
// ===== library types =====

// folder: Library/Modbus/Core/sb

TYPE "mb_station_block_udt"
   STRUCT
      conf : Struct   // Configuration
         skip_code : Bool;   // Skip all code in header and footer fc.
         disable : Bool;   // Skip all queries
         read_only : Bool;   // Skip all write queries. (fc 5,6,15,16)
         max_comm_error : USInt := 2;   // Repeating erros before communication_error flag is set
         exec_x_quries : USInt := 1;   // Number of queries to be exec. at each loop.
      END_STRUCT;
      out : Struct   // Outputs
         error : Bool;   // All errors, including communication errors
         communication_error : Bool;   // only communication errors
         finnish : Bool;   // qid is handed over to next device.
      END_STRUCT;
      log : Struct   // Logging for development and debugging.
         connected_time : DTL;   // The time the device was connected to the bus
         disconnected_time : DTL;   // The time, if a device was disconnected to the bus
         done_cnt : UDInt;   // Successfully queries counter for this device
         error_comm_cnt : UDInt;   // Communication erros cnt.
         error_exception_cnt : UDInt;   // Failed queries counter for this device
         error_status : Word;   // Status code from mb_master or mb_client
         error_data_addr : UDInt;   // d_addr for last failed querie; handy for troubleshooting
      END_STRUCT;
      z : Struct   // Internal states.
         header_qid : UInt;   // qid value at device header
         comm_err_cnt : USInt;   // Repeating communication errors
         exec_cnt : USInt;   // Numb. of exec. q. this loop
         offset_qid : UInt := 1;   // Device query id.
         err_hold : Bool;   // Help var for .out.error
      END_STRUCT;
   END_STRUCT;
END_TYPE

// folder: Library/Modbus/Station blocks/sb untested/Mettler

TYPE "mettlerToledoInd560Udt"
   STRUCT
      readMsgSlot : Array[1..4] of Struct
         cmdRespons : Struct
            FP_1 : Bool;
            FP_2 : Bool;
            FP_3 : Bool;
            FP_4 : Bool;
            FP_5 : Bool;
            data_integrity : Bool;
            cmdAck1 : Bool;
            cmdAck2 : Bool;
         END_STRUCT;
         reserved : Byte;   // volt
         data : Real;
         scale_status : Struct
            x08_Enter_Key : Bool;
            x09_Input_1 : Bool;
            x10_Input_2 : Bool;
            x11_Input_3 : Bool;
            x12_Motion : Bool;
            x13_Net_Mode : Bool;
            x14_Data_Integrity_2 : Bool;
            x15_Data_OK : Bool;
            x00_Target_1 : Bool;
            x01_Comparator_1 : Bool;
            x02_Targe_2 : Bool;
            x03_Comparator_2 : Bool;
            x04_Target_3 : Bool;
            x05_Alway_true : Bool;
            x06_TE_bit_1 : Bool;
            x07_TE_bit_2 : Bool;
         END_STRUCT;
      END_STRUCT;
      writeMsgSlot : Array[1..4] of Struct
         cmd : UInt;
         data : Real;
      END_STRUCT;
      run : Struct   // Data calculated from readMsgSlot
         PF : Array[1..4] of USInt;   // Floating point input indication
         cmdAck : Array[1..4] of USInt;
      END_STRUCT;
      occupiedMsgSlots : Array[1..4] of Bool;
      queryDone : Struct
         read : Bool;
         write : Bool;
      END_STRUCT;
   END_STRUCT;
END_TYPE

// folder: (top level)

FUNCTION_BLOCK "modbus_rtu_1500"   // FB97, LAD
TITLE = Example modbus rtu for S7-1500
{ S7_Optimized_Access := 'TRUE' }
VERSION : 0.1
   VAR
      mb_master_ctrl : "mb_master_1500_ctrl";
      mb_query : "mb_query";
      aquaMaster_device1 : "abb_aquaMaster_3";
      aquaMaster_device2 : "abb_aquaMaster_3";
      Auma_valve : "Auma_valve";
      Phoenix_Contact_UPS : "Phoenix_Contact_UPS";
   END_VAR
   VAR_TEMP   // added for the SCL form of the ladder/FBD networks
      _w1 : Bool;
   END_VAR
BEGIN

REGION Network 1: Modbus master
   // hardware_id:            Can be found inside "Device configuration". Replace hardware_id with correct id.
   // operating_mode:    0: RS232, 2: RS422, 4: RS485.
   // baud:                         Bits per sec. (Parity is even by default)
   // mb_query:                The FB that connects everything together.
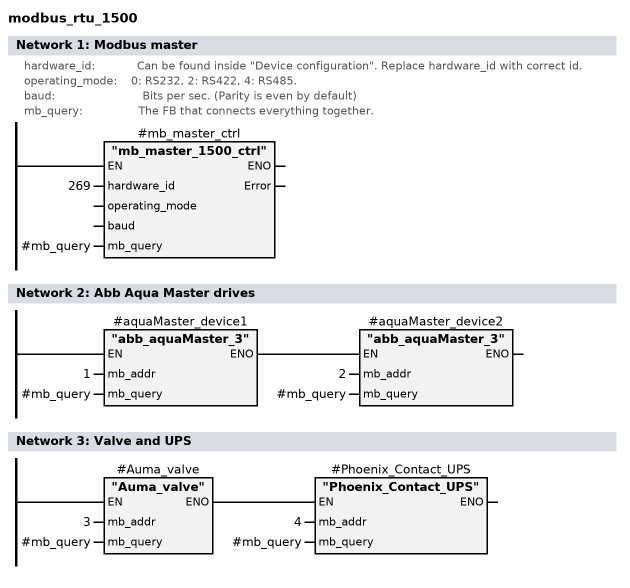
   RUNG wire#powerrail
      #mb_master_ctrl(hardware_id := 269, operating_mode :=, baud :=, mb_query := #mb_query, Error =>)
   END_RUNG
   // the same network as SCL:
   #mb_master_ctrl(hardware_id := 269, mb_query := #mb_query);   // "mb_master_1500_ctrl"
END_REGION

REGION Network 2: Abb Aqua Master drives
   RUNG wire#powerrail
      #aquaMaster_device1(mb_addr := 1, mb_query := #mb_query)
      #aquaMaster_device2(mb_addr := 2, mb_query := #mb_query)
   END_RUNG
   // the same network as SCL:
   #aquaMaster_device1(mb_addr := 1, mb_query := #mb_query, ENO => #_w1);   // "abb_aquaMaster_3"
   IF #_w1 THEN
       #aquaMaster_device2(mb_addr := 2, mb_query := #mb_query);   // "abb_aquaMaster_3"
   END_IF;
END_REGION

REGION Network 3: Valve and UPS
   RUNG wire#powerrail
      #Auma_valve(mb_addr := 3, mb_query := #mb_query)
      #Phoenix_Contact_UPS(mb_addr := 4, mb_query := #mb_query)
   END_RUNG
   // the same network as SCL:
   #Auma_valve(mb_addr := 3, mb_query := #mb_query, ENO => #_w1);   // "Auma_valve"
   IF #_w1 THEN
       #Phoenix_Contact_UPS(mb_addr := 4, mb_query := #mb_query);   // "Phoenix_Contact_UPS"
   END_IF;
END_REGION
END_FUNCTION_BLOCK

FUNCTION_BLOCK "modbus_tcp"   // FB98, LAD
TITLE = Example modbus tcp
{ S7_Optimized_Access := 'TRUE' }
VERSION : 0.1
   VAR
      mb_client_ctrl : "mb_client_ctrl";
      mb_query : "mb_query";
      mb_delay_between_queries : "mb_delay_between_queries";
      ip : Array[1..4] of Byte;
      siemens_PAC3200 : "siemens_PAC3200";
   END_VAR
   VAR_TEMP   // added for the SCL form of the ladder/FBD networks
      _w1 : Bool;
   END_VAR
BEGIN

REGION Network 1 (SCL): IP-address
   #ip[1] := 192;
   #ip[2] := 168;
   #ip[3] := 1;
   #ip[4] := 123;
END_REGION

REGION Network 2: Modbus client ctrl
   // - Insert interface constant, eg "Local~PROFINET_interface_1". 
   // - conn_id need to be unique for the whole plc.
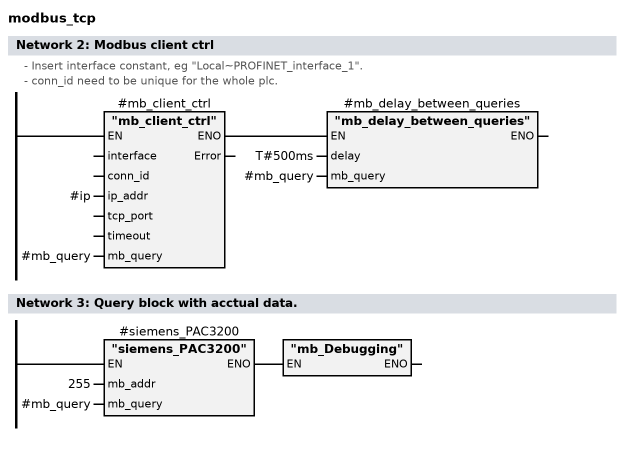
   RUNG wire#powerrail
      #mb_client_ctrl(interface :=, conn_id :=, ip_addr := #ip, tcp_port :=, timeout :=, mb_query := #mb_query, Error =>)
      #mb_delay_between_queries(delay := T#500ms, mb_query := #mb_query)
   END_RUNG
   // the same network as SCL:
   #mb_client_ctrl(ip_addr := #ip, mb_query := #mb_query, ENO => #_w1);   // "mb_client_ctrl"
   IF #_w1 THEN
       #mb_delay_between_queries(delay := T#500ms, mb_query := #mb_query);   // "mb_delay_between_queries"
   END_IF;
END_REGION

REGION Network 3: Query block with acctual data.
   RUNG wire#powerrail
      #siemens_PAC3200(mb_addr := 255, mb_query := #mb_query)
      "mb_Debugging"()
   END_RUNG
   // the same network as SCL:
   #siemens_PAC3200(mb_addr := 255, mb_query := #mb_query, ENO => #_w1);   // "siemens_PAC3200"
   IF #_w1 THEN "mb_Debugging"(); END_IF;
END_REGION
END_FUNCTION_BLOCK

// folder: Library/Modbus/.Start examples

FUNCTION_BLOCK "modbus_rtu_1200"   // FB104, SCL
{ S7_Optimized_Access := 'TRUE' }
VERSION : 0.1
   VAR
      mb_query : "mb_query";
      mb_master_1200_ctrl : "mb_master_1200_ctrl";
      abb_aquaMaster_device1 : "abb_aquaMaster_3";
      abb_aquaMaster_device2 : "abb_aquaMaster_3";
      abb_aquaMaster_device3 : "abb_aquaMaster_3";
      Auma_valve : "Auma_valve";
      Phoenix_Contact_UPS : "Phoenix_Contact_UPS";
      resault_data : Word;
   END_VAR
BEGIN
   // hardware_id: Can be found inside "Device configuration".
   // baud:        Bits per sec. (Parity is even by default)
   // timeout:     Automatically calculated if set to T#0s.
   // mb_query:    The FB that connects everything together.
   #mb_master_1200_ctrl(hardware_id := 0, // REPLACE WITH CORRECT ID.
                        baud := 19200,
                        mb_query := #mb_query);

   // Each blocks bellow represent one device on the bus.

   // Three Abb aqua-master's.
   #abb_aquaMaster_device1(mb_addr := 1, mb_query := #mb_query);
   #abb_aquaMaster_device2(mb_addr := 2, mb_query := #mb_query);
   #abb_aquaMaster_device3(mb_addr := 3, mb_query := #mb_query);

   // A valve 
   #Auma_valve(mb_addr := 4, mb_query := #mb_query);

   // A UPS.
   #Phoenix_Contact_UPS(mb_addr := 5, mb_query := #mb_query);

   // A station block can be used both for both modbus rtu and tcp. This
   // is particular useful if a tcp-rtu-gateway is used. The same program
   // could be used, just swap mb_master_1200_ctrl, with mb_client_ctrl.

   // Read holding register 456 from device with modbus address 123.
   // This is an example showing that a query does not necessarily need
   // to be part of a station block (SB) as obove, however making
   // reusable SB's is good practice.
   #mb_query(mb_addr := 123,
             mode := #mb_query.c.read.holding_reg,
             data_addr := 456,
             data_ptr := #resault_data);


   // Debugging tip, (no code)
   "mb_Debugging"();
END_FUNCTION_BLOCK

FUNCTION_BLOCK "modbus_rtu_1500"   // FB108, SCL
{ S7_Optimized_Access := 'TRUE' }
VERSION : 0.1
   VAR
      mb_query : "mb_query";
      mb_master_1500_ctrl : "mb_master_1500_ctrl";
      abb_aquaMaster_device1 : "abb_aquaMaster_3";
      abb_aquaMaster_device2 : "abb_aquaMaster_3";
      abb_aquaMaster_device3 : "abb_aquaMaster_3";
   END_VAR
BEGIN
   // hardware_id:     May be found inside the hardware configuration.
   // operating_mode:  0: RS232, 2: RS422, 4: RS485.
   // baud:            Bits per sec. (Parity is even by default)
   // timeout:         Automatically calculated if set to zero. (T#0s)
   // mb_query:        The FB that connects everything together.
   #mb_master_1500_ctrl(hardware_id := 0, // REPLACE WITH CORRECT ID.
                        operating_mode := 4, // RS-485
                        baud := 19200, // bps
                        mb_query := #mb_query);

   // Each blocks bellow represent one device on the bus. 
   #abb_aquaMaster_device1(mb_addr := 1, mb_query := #mb_query);
   #abb_aquaMaster_device2(mb_addr := 2, mb_query := #mb_query);
   #abb_aquaMaster_device3(mb_addr := 3, mb_query := #mb_query);


   // Debugging tip, (no code)
   "mb_Debugging"();
END_FUNCTION_BLOCK

FUNCTION_BLOCK "modbus_tcp"   // FB110, SCL
{ S7_Optimized_Access := 'TRUE' }
VERSION : 0.1
   VAR
      mb_query : "mb_query";
      mb_client_ctrl : "mb_client_ctrl";
      siemens_PAC3200 : "siemens_PAC3200";
      ip : Array[1..4] of Byte;
      mb_delay_between_queries : "mb_delay_between_queries";
   END_VAR
BEGIN
   // IP-address of the modbus server
   #ip[1] := 192;
   #ip[2] := 168;
   #ip[3] := 1;
   #ip[4] := 2;

   // interface:  Profinet interface.
   //             (Find const. inside "Device configuration")
   // conn_id:    A unique id for each tcp connectin in the plc.
   // ip_addr:    The ip-address of the server. (Array of 4 bytes)
   // tcp_port:   Default port is 502. (UDP isn't available)
   // timeout:    Depends on the network conncetion.
   // mb_query:   The query FB.
   #mb_client_ctrl(interface := 0, // REPLACE WITH CORRECT ID OR CONST,
                                   // Eg. "Local~PROFINET_interface_1",
                   conn_id := 123,
                   ip_addr := #ip,
                   tcp_port := 502,
                   timeout := T#400ms,
                   mb_query := #mb_query);

   // Delay the query execution, this prevent the plc from
   // jamming the network. Adjust the time to the application.
   #mb_delay_between_queries(delay := T#500ms,
                             mb_query := #mb_query);

   #siemens_PAC3200(mb_query := #mb_query);


   // Debugging tip, (no code)
   "mb_Debugging"();
END_FUNCTION_BLOCK

FUNCTION "mb_Readme" : Void   // FC13, SCL
{ S7_Optimized_Access := 'TRUE' }
VERSION : 0.1
BEGIN
   (* Instructions:

   - Add one of the exmple FB's to your PLC.
   - Call that FB from a cyclic OB.
   - Terminate connection to type on the example FB. (Right click the FB)
   - Set hardware_id, buad-rate, ip, tcp-port, etc, to the correct value.
   - Look inside the library and check if there is a ready station block (SB),
     for your program. If there isn't then a new has to be made. 
   - Station blocks can be single-DB's or multi-instances in a FB.
   - Remove the exmple code and example SB's.

   IMPORTANT: As stated above, the start examples fb, need to be terminated 
              from it's type. If the type is edited and later there is a 
              library update, then all the changes will get lost.

   - Instructions need to be of the latest version, 
     this is usually already set:
      * Instructions -> Communication -> Others -> Modbus TCP
      * Instructions -> Communication -> Communication processor -> Modbus
      * Instructions -> Communication -> Communication processor -> Modbus (RTU)  
      * Instructions -> Basic instructions -> Word logic operations -> SEL.
     Change version in the right column.

   *)
END_FUNCTION

// folder: Library/Modbus/.Start examples/Empty

FUNCTION_BLOCK "modbus_rtu_1500"   // FB5, SCL
{ S7_Optimized_Access := 'TRUE' }
VERSION : 0.1
   VAR
      mb_query : "mb_query";
      mb_master_1500_ctrl : "mb_master_1500_ctrl";
      _ : Bool;
   END_VAR
BEGIN
   // hardware_id:     May be found inside the hardware configuration.
   // operating_mode:  0: RS232, 2: RS422, 4: RS485.
   // baud:            Bits per sec. (Parity is even by default)
   // timeout:         Automatically calculated if set to zero. (T#0s)
   // mb_query:        The FB that connects everything together.
   #mb_master_1500_ctrl(hardware_id := 0, // REPLACE WITH CORRECT ID.
                        operating_mode := 4, // RS-485
                        baud := 19200, // bps
                        mb_query := #mb_query);





   // Debugging tip, (no code)
   "mb_Debugging"();
END_FUNCTION_BLOCK

FUNCTION_BLOCK "modbus_tcp"   // FB79, SCL
{ S7_Optimized_Access := 'TRUE' }
VERSION : 0.1
   VAR
      mb_query : "mb_query";
      mb_client_ctrl : "mb_client_ctrl";
      ip : Array[1..4] of Byte;
      mb_delay_between_queries : "mb_delay_between_queries";
   END_VAR
BEGIN
   // IP-address of the modbus server
   #ip[1] := 192;
   #ip[2] := 168;
   #ip[3] := 1;
   #ip[4] := 2;

   // interface:  Profinet interface.
   //             (Find const. inside "Device configuration")
   // conn_id:    A unique id for each tcp connectin in the plc.
   // ip_addr:    The ip-address of the server. (Array of 4 bytes)
   // tcp_port:   Default port is 502. (UDP isn't available)
   // timeout:    Depends on the network conncetion.
   // mb_query:   The query FB.
   #mb_client_ctrl(interface := 0, // REPLACE WITH CORRECT ID OR CONST,
                                   // Eg. "Local~PROFINET_interface_1",
                   conn_id := 123,
                   ip_addr := #ip,
                   tcp_port := 502,
                   timeout := T#400ms,
                   mb_query := #mb_query);

   // Delay the query execution, this prevent the plc from
   // jamming the network. Adjust the time to the application.
   #mb_delay_between_queries(delay := T#500ms,
                             mb_query := #mb_query);






   // Debugging tip, (no code)
   "mb_Debugging"();
END_FUNCTION_BLOCK

FUNCTION_BLOCK "modbus_rtu_1200"   // FB111, SCL
{ S7_Optimized_Access := 'TRUE' }
VERSION : 0.1
   VAR
      mb_query : "mb_query";
      mb_master_1200_ctrl : "mb_master_1200_ctrl";
      _ : Bool;
   END_VAR
BEGIN
   // hardware_id: Can be found inside "Device configuration".
   // baud:        Bits per sec. (Parity is even by default)
   // timeout:     Automatically calculated if set to T#0s.
   // mb_query:    The FB that connects everything together.
   #mb_master_1200_ctrl(hardware_id := 0, // REPLACE WITH CORRECT ID. ("Local~CB_1241_(RS485)")
                        baud := 19200,
                        mb_query := #mb_query);





   // Debugging tip, (no code)
   "mb_Debugging"();
END_FUNCTION_BLOCK

// folder: Library/Modbus/.Start examples/Ladder

FUNCTION_BLOCK "modbus_rtu_1200"   // FB97, LAD
TITLE = Example modbus rtu
{ S7_Optimized_Access := 'TRUE' }
VERSION : 0.1
// REPLACE hardware_id WITH CORRECT ID.
   VAR
      mb_master_ctrl : "mb_master_1200_ctrl";
      mb_query : "mb_query";
      aquaMaster_device1 : "abb_aquaMaster_3";
      aquaMaster_device2 : "abb_aquaMaster_3";
      Auma_valve : "Auma_valve";
      Phoenix_Contact_UPS : "Phoenix_Contact_UPS";
   END_VAR
   VAR_TEMP   // added for the SCL form of the ladder/FBD networks
      _w1 : Bool;
   END_VAR
BEGIN

REGION Network 1: Modbus master
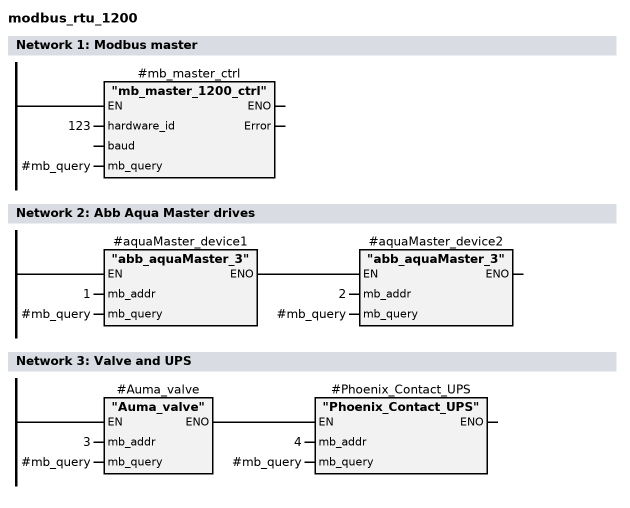
   RUNG wire#powerrail
      #mb_master_ctrl(hardware_id := 123, baud :=, mb_query := #mb_query, Error =>)
   END_RUNG
   // the same network as SCL:
   #mb_master_ctrl(hardware_id := 123, mb_query := #mb_query);   // "mb_master_1200_ctrl"
END_REGION

REGION Network 2: Abb Aqua Master drives
   RUNG wire#powerrail
      #aquaMaster_device1(mb_addr := 1, mb_query := #mb_query)
      #aquaMaster_device2(mb_addr := 2, mb_query := #mb_query)
   END_RUNG
   // the same network as SCL:
   #aquaMaster_device1(mb_addr := 1, mb_query := #mb_query, ENO => #_w1);   // "abb_aquaMaster_3"
   IF #_w1 THEN
       #aquaMaster_device2(mb_addr := 2, mb_query := #mb_query);   // "abb_aquaMaster_3"
   END_IF;
END_REGION

REGION Network 3: Valve and UPS
   RUNG wire#powerrail
      #Auma_valve(mb_addr := 3, mb_query := #mb_query)
      #Phoenix_Contact_UPS(mb_addr := 4, mb_query := #mb_query)
   END_RUNG
   // the same network as SCL:
   #Auma_valve(mb_addr := 3, mb_query := #mb_query, ENO => #_w1);   // "Auma_valve"
   IF #_w1 THEN
       #Phoenix_Contact_UPS(mb_addr := 4, mb_query := #mb_query);   // "Phoenix_Contact_UPS"
   END_IF;
END_REGION
END_FUNCTION_BLOCK

// folder: Library/Modbus/Core

FUNCTION_BLOCK "mb_query"   // FB1, SCL
{ S7_Optimized_Access := 'TRUE' }
VERSION : 0.1
   VAR_INPUT
      mb_addr : UInt;   // Device addr. (0 to 247)
      mode : USInt;   // Function code: 1,2,3,4,5,6,15,16. (siemens mode shifted to 200 - 202)
      data_addr : UDInt;   // Data addr. (raw telegram value, 0-65535)
      data_len : UInt;   // Data len. 0=>Auto detect
   END_VAR
   VAR_OUTPUT
      Done : Bool;   // Successful query
      Error : Bool;   // Failed query
   END_VAR
   VAR_IN_OUT
      data_ptr : Variant;   // Bytes and bools has to add up to whole word(s)
   END_VAR
   VAR
      c : Struct   // Constants
         read : Struct   // Read: 1, 2, 3, 4
            discrete_output : USInt := 1;   // 1 (coils)
            discrete_input : USInt := 2;   // 2
            holding_reg : USInt := 3;   // 3
            input_reg : USInt := 4;   // 4
         END_STRUCT;
         write : Struct   // Write: 5, 6, 15, 16
            single_discrete_output : USInt := 5;   // 5 (coil) (when len. is eq. to 1)
            single_holding_reg : USInt := 6;   // 6 (when len. is eq. to 1)
            discrete_output : USInt := 15;   // 15 (coils)
            holding_reg : USInt := 16;   // 16
         END_STRUCT;
         mode : Struct   // Modicon convention addressing. (Eg: hold.reg. start at 40001)
            read : USInt := 200;   // Mode 0 (fc: 1, 2, 3, 4)
            write_single : USInt := 201;   // Mode 1 (fc: 5, 6) (when len. is eq. to 1)
            write : USInt := 202;   // Mode 2 (fc: 15, 16)
         END_STRUCT;
         auto_len : USInt := 0;   // Length based on data_ptr (Used for data_len)
      END_STRUCT;
      conf : Struct   // Configuration
         buffer_handler : Bool := TRUE;   // enable buffer handler
         halt : Bool;   // Halt exec. of queries.
      END_STRUCT;
      stat : Struct   // Status of last executed query
         done : Bool;   // Successfull
         error : Bool;   // Error, including timeout error
         busy : Bool;   // mb_master or mb_client is busy.
         error_comm : Bool;   // communication error (timeout or bad crc)
         status : Word;   // status word of mb_master or mb_client
      END_STRUCT;
      z : Struct   // Internal states
         q : Struct   // Query params
            mb_addr : UInt := 1;   // Station address
            mode : USInt := 0;   // Function code
            data_addr : UDInt;   // Data address
            data_len : UInt := 0;   // Data length
         END_STRUCT;
         run : Struct   // Constantly changing variables
            qid : UInt := 1;   // query id
            qid_cnt : UInt;   // Query id cnt. increase for each query, reset in controller. One loop each scan
            state : USInt;
            write : Bool;   // A write query is inserted
            discrete : Bool;
         END_STRUCT;
         sb : Struct   // Station block functionality
            sid : UInt;   // Device ID
            sid_halt : Bool;
            sid_cnt : UInt;   // Device id cnt
            sid_retry : UInt := 1;   // Retry device id, qComError
            sid_retry_finished : Bool;
            seq_release : Bool;
            head_insert : Bool;   // Inc. at mb_query on insert
            head_recive : Bool;   // Inc. at mb_query on rec.
            reset : Bool;
            log_data_addr : UDInt;   // Tmp.var. for transf. value to mb_device_footer
         END_STRUCT;
         buffer : Array[0..249] of Byte;
      END_STRUCT;
   END_VAR
   VAR_TEMP
      tLen : UInt;
      tPos : DInt;
      tDiscrete : Bool;
      "e" : Int;
      tBuffer : Array[0..249] of Byte;
   END_VAR
   VAR CONSTANT
      ORIGIN : USInt := 0;
      INSERT_QUERY : USInt := 1;
      INIT_QUERY : USInt := 2;
      EXEC_QUERY : USInt := 3;
      RECIVE_RESUALT : USInt := 4;
   END_VAR
BEGIN
   // Rexhip - Extended modbus library 
   // --- --- --- ---
   // License:  MIT-license
   // Author:   Ola Bjørnli
   // Web:      www.rexhip.com
   //           github.com/rexhip/rexhip
   // --- --- --- ---
   // 
   // For autmatic calculation of data_len, mb_query can only count whole
   // words (16 bits). This implices that the automatic length works well
   // for holding- and input registers, but dosen't work for dicreate
   // queries. For this queries data_len need to be specified manually.
   // After a query where data_len is specified, it need to be set back
   // to automatic. (#mb_query.data_len := #mb_query.c.auto_len;)
   //
   // Please read to the documentation and see the examples, before dive
   // into the code bellow.

   REGION Header            
       #Done := #Error := false;

       // qid_cnt is increased for every query (above) and reset back
       // to zero in mb_internal_e. Qid (query id) is increased when a
       // query finnish. A query will execute when qit_cnt = qid. Qid
       // is set back to "1" when all queryies has been executed.
       #z.run.qid_cnt += 1;
       IF #z.run.qid_cnt <> #z.run.qid
           OR #stat.busy // mb_master.busy or mb_client.busy
       THEN
           RETURN;
       END_IF;
   END_REGION

   REGION Pre-calc
       // Is this a discrete query ?
       CASE #mode OF
           1, 2, 5, 15: // Function codes
               #tDiscrete := true;
           200..202:
               CASE #data_addr OF
                   1..19999: // 1..9999, 10001..19999:
                       #tDiscrete := true;
               END_CASE;
       END_CASE;

       // data_len=0 => Automatically calculate the length.
       IF #data_len = 0 THEN
           #"e" := Serialize(SRC_VARIABLE := #data_ptr,
                           DEST_ARRAY => #tBuffer,
                           POS := #tPos);
           #tLen := DINT_TO_UINT
           (* *)(SEL(G := #tDiscrete, IN0 := #tPos / 2, IN1 := #tPos * 8));
       ELSE
           #tLen := #data_len;
       END_IF;
   END_REGION

   // Wait inserting next query if halted, else just continue.
   IF #z.run.state = #ORIGIN AND NOT #conf.halt THEN
       #z.run.state := #INSERT_QUERY;
   END_IF;

   CASE #z.run.state OF
       #INSERT_QUERY: // Transfer query params. to internal variables.

           // Figur out if this is a query that will write to the device.
           CASE #mode OF
               5, 6, 15, 16, 201, 202: // Write fc's.
                   #z.run.write := true;
               ELSE // Read
                   #z.run.write := false;
           END_CASE;

           #z.run.discrete := #tDiscrete;

           // The params is transfered over to the internal mem. They
           // are later transfered to the modbus master block or the
           // client block.
           #z.q.mb_addr := #mb_addr;
           #z.q.mode := #mode;
           #z.q.data_addr := #data_addr;
           #z.q.data_len := #tLen;

           IF #conf.buffer_handler AND #z.run.write THEN
               // Copy the content of #data_ptr to the buffer.
               #tPos := 0; // Start at the beginning of the buffer.
               #"e" := Serialize(SRC_VARIABLE := #data_ptr,
                               DEST_ARRAY => #z.buffer,
                               POS := #tPos);
           END_IF;
           // A msg. to station block foother FC, a new query has
           // been inserted.
           #z.sb.head_insert := true;

           #z.run.state := #INIT_QUERY; // State inside ctrl block.


       #RECIVE_RESUALT: // Query is finnished. (with or without error)  

           // Make sure that the query resault really belong to this
           // query. This may not be the case if another query before
           // is surrounded by a if-statement.
           IF #z.q.mb_addr = #mb_addr
               AND #z.q.mode = #mode
               AND #z.q.data_addr = #data_addr
               AND #z.q.data_len = #tLen
           THEN
               IF #stat.done // Successfull query (no error)
                   AND NOT #z.run.write  // If it's a read query.
                   AND #conf.buffer_handler
               THEN
                   // Copy the content from the buffer to #data_ptr
                   #tPos := 0; // Start at the beginning of the buffer.
                   #"e" := Deserialize(SRC_ARRAY := #z.buffer,
                                     DEST_VARIABLE => #data_ptr,
                                     POS := #tPos);
               END_IF;
               #Done := #stat.done;
               #Error := #stat.error;

               // Temperary store value, so it can be picked up
               // in the sb footer.
               #z.sb.log_data_addr := #data_addr;
               // Msg. to mb_station_footer.
               #z.sb.head_recive := true;
           END_IF;
           #z.run.qid += 1; // Next query
           #z.run.state := #ORIGIN; // (State before insert, see above)
   END_CASE;
END_FUNCTION_BLOCK

FUNCTION "mb_version" : String   // FC6, SCL
{ S7_Optimized_Access := 'TRUE' }
VERSION : 0.1
BEGIN
   // Library version.
   #mb_version := '3.1.0';

   (*
   License: MIT-license 
   (https://github.com/rexhip/rexhip/blob/master/docs/License.txt)

   www.rexhip.com
   github.com/rexhip/rexhip


   Author: Ola Bjørnli 

   *)
END_FUNCTION

// folder: Library/Modbus/Core/Ctrl

FUNCTION_BLOCK "mb_client_ctrl"   // FB9, SCL
{ S7_Optimized_Access := 'TRUE' }
VERSION : 1.0
   VAR_INPUT
      interface : Hw_Any := 64;   // Profinet interface id
      conn_id : Conn_Ouc := 123;   // Connection id. Should be unique between all tcp connections.
      ip_addr : Array[1..4] of Byte;   // IPv4 address.
      tcp_port : UInt := 502;   // TCP port
      timeout : Time := T#2s;
   END_VAR
   VAR_OUTPUT
      Error : Bool;   // error flag with tof timer
   END_VAR
   VAR_IN_OUT
      mb_query : "mb_query";   // udt mb
   END_VAR
   VAR
      conf : Struct   // Configuration that normal shouldn't need to be changed.
         disconnect : Bool := FALSE;
         retries : USInt := 1;
         timeout_connect : Time;   // May be set longer, then the main timeout. T#0s => Use normal timeout.
         disconnect_on_80A3 : Bool := true;
      END_STRUCT;
      client : MB_CLIENT;
      tdiscon : TDISCON;
      tcon_ip_v4 : TCON_IP_v4;
      ton_connect : TON_TIME;
      end : "mb_internal_e";
      connected_least_once : Bool;   // One connection has taken place.
   END_VAR
   VAR_TEMP
      comm_err : Bool;
   END_VAR
   VAR CONSTANT
      INIT_QUERY : USInt := 2;
      EXEC_QUERY : USInt := 3;
      RECIVE_RESUALT : USInt := 4;
   END_VAR
BEGIN
   // Rexhip - Extended modbus library.
   // Please see top section of mb_query for more info.
   //
   // Modbus tcp for S7-1200 and S7-1500.

   REGION Init
       #tcon_ip_v4.InterfaceId := #interface;
       #tcon_ip_v4.ID := #conn_id;
       #tcon_ip_v4.ConnectionType := 11; // tcp
       #tcon_ip_v4.ActiveEstablished := true;
       #tcon_ip_v4.RemoteAddress.ADDR := #ip_addr;
       #tcon_ip_v4.RemotePort := #tcp_port;

       PRESET_TIMER(PT :=
                    SEL(G := #conf.timeout_connect = T#0s
                        OR NOT #connected_least_once,
                        IN0 := #conf.timeout_connect,
                        IN1 := #timeout),
                    TIMER := #ton_connect);
       #ton_connect(IN := NOT #conf.disconnect AND NOT #client.Connected,
                    PT := #ton_connect.PT);
       // - Use #timeout if: #timeout_connect is set to zero, or there has
       //   been a least one connection to the server.
       // - Establing a TCP connection may take long. 
       // - If mb_client does not establish a connection it will not  throw
       //   timeout error. Timeout is handled manually for that case. 

       // Conversion of function codes. 
       IF #mb_query.z.run.state = #INIT_QUERY THEN
           CASE #mb_query.z.q.mode OF
               1..16: // 1..6, 15, 16:
                   #client.MB_MODE := #mb_query.z.q.mode + 100;
                   // Eg. Siemens use 103 for fc 3. (read halding reg)
               200..202:
                   #client.MB_MODE := #mb_query.z.q.mode - 200;
               ELSE
                   #client.MB_MODE := #mb_query.z.q.mode;
           END_CASE;
           #client.MB_Unit_ID := UINT_TO_BYTE(#mb_query.z.q.mb_addr);
           #client.Retries := #conf.retries;
           #mb_query.z.run.state := #EXEC_QUERY; // Next state.
       END_IF;
   END_REGION

   REGION Exec
       // STATUS 16#80A3 : 
       // If a new download has taken place, and this block is re-initialize,
       // then the mb_client block will output the error code saying that:
       // "Attempt being made to re-establish an existing connection." The
       // solution to this problem is to disconnect and then reconnect. It
       // dosen't work to use disconnect input on the mb_client block.
       #tdiscon(REQ := #client.STATUS = 16#80A3 AND #conf.disconnect_on_80A3,
                ID := #conn_id);

       #client.Rcv_Timeout :=
       (* *)UDINT_TO_REAL(T_CONV(#timeout)) * 0.001; // ms to s.
       #client(DISCONNECT := #conf.disconnect OR #tdiscon.BUSY,
               REQ := #mb_query.z.run.state = #EXEC_QUERY
               AND NOT #client.BUSY
               AND NOT #client.DISCONNECT,
               MB_MODE := #client.MB_MODE,
               MB_DATA_ADDR := #mb_query.z.q.data_addr,
               MB_DATA_LEN := #mb_query.z.q.data_len,
               BUSY => #mb_query.stat.busy,
               MB_DATA_PTR := #mb_query.z.buffer,
               CONNECT := #tcon_ip_v4);

       IF #mb_query.z.run.state = #EXEC_QUERY THEN
           #mb_query.stat.error := #client.ERROR OR #ton_connect.Q;
           #mb_query.stat.done := #client.DONE AND NOT #mb_query.stat.error;
           #mb_query.stat.status := #client.STATUS;
           // Comm. error and timeout handeling. 
           CASE WORD_TO_UINT(#mb_query.stat.status) OF
               16#80C8,  // No response from the server.
               16#818C: // blocked_proc_timeout or rcv_timeout.
                   #comm_err := #mb_query.stat.error;
           END_CASE;
           #mb_query.stat.error_comm := #ton_connect.Q OR #comm_err;
       END_IF;
   END_REGION

   // End is a comman FB for both tcp and rtu.
   #end(mb_query := #mb_query, Error => #Error);
END_FUNCTION_BLOCK

FUNCTION_BLOCK "mb_master_1500_ctrl"   // FB10, SCL
{ S7_Optimized_Access := 'TRUE' }
VERSION : 1.0
   VAR_INPUT
      hardware_id : Port;   // hardware id
      operating_mode : USInt := 4;   // 0: RS232, 2: RS422, 4: RS485.
      baud : UDInt := 19200;   // Bits per sec.
   END_VAR
   VAR_OUTPUT
      Error : Bool;   // One or more errors in the whole application.
   END_VAR
   VAR_IN_OUT
      mb_query : "mb_query";
   END_VAR
   VAR
      conf : Struct   // Configuration that normal shouldn't need to be changed.
         parity : UInt := 2;   // 0=no-parity, 1=odd, 2=even.
         retries : USInt := 0;
         timeout : Time;   // Automatically calculated if set to zero. (T#0s)
      END_STRUCT;
      comm_load : Modbus_Comm_Load;
      master : Modbus_Master;
      buffer : "mb_internal_b";
      end : "mb_internal_e";
      comm_load_done : Bool;
      init_hw : Bool := true;
   END_VAR
   VAR CONSTANT
      INIT_QUERY : USInt := 2;
      EXEC_QUERY : USInt := 3;
      RECIVE_RESUALT : USInt := 4;
   END_VAR
BEGIN
   // Rexhip - Extended modbus library.
   // Please see top section of mb_query for more info.
   //
   // RTU master for S7-1500
   // 
   // This master blocks works for both S7-1200 and S7-1500. For S7-1200
   // it's recommended to use the other master block, mb_master_1200_ctrl
   // because it use less memory. Please read the documentation, before
   // dive into the code bellow.

   REGION Init
       IF #init_hw THEN
           // T#0s => Automatically adjust timeout.
           #comm_load.RESP_TO :=
           SEL(G := #conf.timeout = T#0s,
               IN0 := T_CONV(#conf.timeout),
               IN1 := UDINT_TO_UINT(4500000 / #baud));
       END_IF;
       // Initiate the hardware.
       #comm_load.RETRIES := #conf.retries;
       #comm_load.MODE := #operating_mode;
       #comm_load(REQ := #init_hw,
                  PORT := #hardware_id,
                  BAUD := #baud,
                  PARITY := #conf.parity, // Even is default.
                  RESP_TO := #comm_load.RESP_TO,
                  MB_DB := #master.MB_DB);
       #init_hw := false; // Hw init Finnised
       IF #comm_load.DONE THEN
           #comm_load_done := true;
       END_IF;

       IF #mb_query.z.run.state = #INIT_QUERY THEN
           // Modicon convention address conversion.
           "mb_internal_a"(mode104 := true,
                          Mode => #master.MODE,
                          Data_addr => #master.DATA_ADDR,
                          mb_query := #mb_query);

          // Copy buffer to a non optimiced memory area.
           IF #mb_query.z.run.write THEN
               #buffer.buffer := #mb_query.z.buffer;
           END_IF;

           IF #comm_load_done THEN
               #mb_query.z.run.state := #EXEC_QUERY;
           ELSE
               // Skip query exec. if init hw didn't go well.
               // The state RECIVE_RESUALT is inside mb_query.
               #mb_query.z.run.state := #RECIVE_RESUALT;
               #mb_query.stat.done := false;
               #mb_query.stat.error := true;
               #mb_query.stat.error_comm := true;
               #mb_query.stat.status := #comm_load.STATUS;
           END_IF;
       END_IF;
   END_REGION

   REGION Exec
       #master(REQ := #mb_query.z.run.state = #EXEC_QUERY
               AND NOT #master.BUSY,
               MB_ADDR := #mb_query.z.q.mb_addr,
               MODE := #master.MODE,
               DATA_ADDR := #master.DATA_ADDR,
               DATA_LEN := #mb_query.z.q.data_len,
               BUSY => #mb_query.stat.busy,
               DATA_PTR := #buffer.buffer);

       IF #mb_query.z.run.state = #EXEC_QUERY THEN
           #mb_query.stat.error := #master.ERROR;
           #mb_query.stat.done := #master.DONE;
           #mb_query.stat.status := #master.STATUS;
           "mb_internal_f"(buffer := #buffer, mb_query := #mb_query);
       END_IF;
   END_REGION

   // End is a comman FB for both tcp and rtu.
   #end(mb_query := #mb_query, Error => #Error);
END_FUNCTION_BLOCK

FUNCTION_BLOCK "mb_master_1200_ctrl"   // FB90, SCL
{ S7_Optimized_Access := 'TRUE' }
VERSION : 1.0
   VAR_INPUT
      hardware_id : Port := 0;   // Hardware id
      baud : UDInt := 19200;   // Bits per second
   END_VAR
   VAR_OUTPUT
      Error : Bool;   // One or more errors in the whole application.
   END_VAR
   VAR_IN_OUT
      mb_query : "mb_query";
   END_VAR
   VAR
      conf : Struct   // Configuration that normal shouldn't need to be changed.
         parity : UInt := 2;   // 0=no-parity, 1=odd, 2=even.
         retries : USInt := 0;
         timeout_gain : Real := 2.0;   // Multiplied with the calculated value.
         timeout_offset : Time := T#0ms;   // Added to the calculated value.
      END_STRUCT;
      comm_load : MB_COMM_LOAD;
      master : MB_MASTER;
      buffer : "mb_internal_b";
      end : "mb_internal_e";   // FB common for both rtu and tcp.
   END_VAR
   VAR_TEMP
      tmp_err : Bool;
   END_VAR
   VAR CONSTANT
      INIT_QUERY : USInt := 2;
      EXEC_QUERY : USInt := 3;
      RECIVE_RESUALT : USInt := 4;
   END_VAR
BEGIN
   // Rexhip - Extended modbus library.
   // Please see top section of mb_query for more info.
   // 
   // RTU master for S7-1200
   // 
   // This FB use less memory then mb_master_1500_ctrl, but it only works for
   // S7-1200 PLC's. Please read the documentation, before dive into the code
   // bellow. See link in mb_query() FB.

   REGION Init
       IF #mb_query.z.run.state = #INIT_QUERY THEN
           // Modicon convention address conversion.
           "mb_internal_a"(mode104 := false,
                          Mode => #master.MODE,
                          Data_addr => #master.DATA_ADDR,
                          mb_query := #mb_query);
           // Copy buffer to a non optimiced memory area.
           IF #mb_query.z.run.write THEN
               #buffer.buffer := #mb_query.z.buffer;
           END_IF;
           // Automatically adjust timeout.
           #comm_load.RESP_TO := T_CONV
           (* *)("mb_timeout_rtu_calc"
                 (**)(gain := #conf.timeout_gain, 
                 (**) offset := #conf.timeout_offset,
                 (**) baud := #baud, mb_query := #mb_query));
           #comm_load.RETRIES := #conf.retries;
       END_IF;

       // Initiate the hardware
       #comm_load(REQ := #mb_query.z.run.state = #INIT_QUERY,
                  PORT := #hardware_id,
                  BAUD := #baud,
                  PARITY := #conf.parity, // Even is default.
                  RESP_TO := #comm_load.RESP_TO,
                  MB_DB := #master);

       IF #mb_query.z.run.state = #INIT_QUERY THEN
           IF #comm_load.DONE THEN
               #mb_query.z.run.state := #EXEC_QUERY;
           ELSE
               // Skip query exec. if init hw didn't go well.
               // The state RECIVE_RESUALT is inside mb_query.
               #mb_query.z.run.state := #RECIVE_RESUALT;
               #mb_query.stat.done := false;
               #mb_query.stat.error := true;
               #mb_query.stat.error_comm := true;
               #mb_query.stat.status := #comm_load.STATUS;
           END_IF;
       END_IF;
   END_REGION

   REGION Exec
       // The core master block.
       #master(REQ := #mb_query.z.run.state = #EXEC_QUERY
               AND NOT #master.BUSY,
               MB_ADDR := #mb_query.z.q.mb_addr,
               MODE := #master.MODE,
               DATA_ADDR := #master.DATA_ADDR,
               DATA_LEN := #mb_query.z.q.data_len,
               BUSY => #mb_query.stat.busy,
               DATA_PTR := #buffer.buffer);

       IF #mb_query.z.run.state = #EXEC_QUERY THEN
           #mb_query.stat.error := #master.ERROR;
           #mb_query.stat.done := #master.DONE;
           #mb_query.stat.status := #master.STATUS;
           "mb_internal_f"(buffer := #buffer, mb_query := #mb_query);
       END_IF;
   END_REGION

   // End is a comman FB for both tcp and rtu.
   #end(mb_query := #mb_query, Error => #Error);
END_FUNCTION_BLOCK

// folder: Library/Modbus/Core/Special

FUNCTION_BLOCK "mb_delay"   // FB11, SCL
{ S7_Optimized_Access := 'TRUE' }
VERSION : 0.1
   VAR_INPUT
      delay : Time;
   END_VAR
   VAR_IN_OUT
      mb_query : "mb_query";
   END_VAR
   VAR
      "timer" : TON_TIME;
      halt : Bool;
   END_VAR
BEGIN
   // For use with modbus tcp, so the client dosen't jam a network.
   // The function halt execution of queries for a certain time

   #mb_query.z.run.qid_cnt += 1;  // The timer occupy one qid.

   IF #halt // If the timer has been activated.
       OR #delay = T#0s // #delay = T#0s => Disable function
   THEN
       PRESET_TIMER(PT := #delay, TIMER := #"timer");
       #"timer"(IN := #delay <> T#0s, PT := #delay);
       IF #"timer".Q OR #delay = T#0s THEN
           IF #halt THEN
               #mb_query.conf.halt := #halt := false; // Continue exec.
               RESET_TIMER(#"timer");
           END_IF;
           #mb_query.z.run.qid += BOOL_TO_UINT
           (* *)(#mb_query.z.run.qid = #mb_query.z.run.qid_cnt);
       END_IF;

   ELSIF #mb_query.z.run.qid_cnt = #mb_query.z.run.qid THEN
       #mb_query.conf.halt := #halt := true; // Halt exec.
   END_IF;
END_FUNCTION_BLOCK

FUNCTION_BLOCK "mb_delay_between_queries"   // FB13, SCL
{ S7_Optimized_Access := 'TRUE' }
VERSION : 0.1
   VAR_INPUT
      delay : Time;
   END_VAR
   VAR_IN_OUT
      mb_query : "mb_query";
   END_VAR
   VAR
      "timer" : TON_TIME;
      halt : Bool;
      old_state : UInt;
   END_VAR
   VAR CONSTANT
      ORIGIN : USInt := 0;
   END_VAR
BEGIN
   // For use with modbus tcp, so the client dosen't jam a network.
   // The function halt execution of queries for a certain time
   // not just once, but between every query. There should only be
   // one of this block for each client.

   IF #halt // Is exec. halted?
       OR #delay = T#0s // #delay = T#0s => Disable function.
   THEN
       PRESET_TIMER(PT := #delay, TIMER := #"timer");
       #"timer"(IN := #delay <> T#0s, PT := #delay);
       IF #"timer".Q
           OR #delay = T#0s AND #halt
       THEN
           RESET_TIMER(#"timer");
           #mb_query.conf.halt := #halt := false; // Continue exec.
       END_IF;

   ELSIF #mb_query.z.run.state <> #old_state
       AND #mb_query.z.run.state <> #ORIGIN
   THEN
       // Halt exec. when next query is about to be inserted,
       // but current query will still finish.
       #mb_query.conf.halt := #halt := true; // Halt exec.
   END_IF;
   #old_state := #mb_query.z.run.state;
END_FUNCTION_BLOCK

FUNCTION "mb_dataptr_eq_buffer" : Bool   // FC3, SCL
{ S7_Optimized_Access := 'TRUE' }
VERSION : 0.1
   VAR_IN_OUT
      data_ptr : Variant;
      mb_query : "mb_query";
   END_VAR
   VAR_TEMP
      tmp_buffer : Array[0..249] of Byte;
      pos : DInt;
      c : Int;
      "e" : Int;
   END_VAR
BEGIN
   // Most use cases will not need this function !
   // Example:
   // 
   // #mb_query(mb_addr := 123,
   //           mode := #mb_query.c.write.holding_reg,
   //           data_addr := 456,
   //           data_ptr := #data);
   //
   // IF #mb_query.Done AND
   //     "mb_dataPtr_eq_buffer"(data_ptr := #data, mb_query := #mb_query)
   // THEN
   //      // If there are for some reason two write queries that has exatly
   //      // the same parameters, then the Done-flag may not be enough to
   //      // determine which query has been executed. To compare data as
   //      // well, data_ptr to the buffer, then this use this function. It
   //      // will return true if the content is the same.
   // END_IF;
   //
   // ------- 

   #mb_dataptr_eq_buffer := true; // Init. value

   #"e" := Serialize(SRC_VARIABLE := #data_ptr,
                   DEST_ARRAY => #tmp_buffer,
                   POS := #pos);

   // Looking for differences.
   FOR #c := 0 TO #pos - 1 DO
       IF #tmp_buffer[#c] <> #mb_query.z.buffer[#c] THEN
           #mb_dataptr_eq_buffer := false;
           EXIT;
       END_IF;
   END_FOR;
END_FUNCTION

FUNCTION "mb_query_bits" : Void   // FC9, SCL
{ S7_Optimized_Access := 'TRUE' }
VERSION : 0.1
   VAR_IN_OUT
      data_ptr : Array[*] of Bool;
      mb_query : "mb_query";
   END_VAR
   VAR_TEMP
      discrete : Bool;
      dommy : Bool;
      lower : DInt;
      upper : DInt;
      bits : UInt;
      bytes : UDInt;   // bytes
   END_VAR
   VAR CONSTANT
      INIT_QUERY : USInt := 2;
      RECIVE_RESUALT : USInt := 4;
   END_VAR
BEGIN
   // This function may be used when the number of bits dosen't
   // add up to whole bytes, for function codes: 1, 2, 5 and 15. 
   // 
   // data_ptr need to be a one dimensional array of bools.
   // --- --- ---

   REGION Header
       IF #mb_query.z.run.qid_cnt + 1 <> #mb_query.z.run.qid
           OR #mb_query.stat.busy
       THEN
           // Skip query, qid will not match qid_cnt and
           // my_query will return.
           #mb_query(data_ptr := #dommy);
           RETURN;
       END_IF;
   END_REGION

   REGION Pre-calc
       // Some preparing calculations.
       CASE #mb_query.mode OF // A discrete query ?
           1, 2, 5, 15:
               #discrete := true;
           200..202:
               CASE #mb_query.data_addr OF
                   1..19999: // 1..9999, 10001..19999
                       #discrete := true;
               END_CASE;
       END_CASE;
       #lower := LOWER_BOUND(ARR := #data_ptr, DIM := 1);
       #upper := UPPER_BOUND(ARR := #data_ptr, DIM := 1);
       #bits := DINT_TO_UINT(#upper - #lower + 1); // Elements in array.

       // Auto data len ?
       IF #mb_query.data_len = #mb_query.c.auto_len THEN
           #bytes := (#bits + 7) / 8; // CEIL()
           #mb_query.data_len := SEL(G := #discrete,
                                     IN0 := (#bits + 15) / 16, // CEIL()
                                     IN1 := #bits);
       ELSE
           #bytes := SEL(G := #discrete,
                         IN0 := #mb_query.data_len * 2, // 1 word -> 2 bytes
                         IN1 := (#mb_query.data_len + 7) / 8); // CEIL()
       END_IF;
   END_REGION

   REGION Run
       // Disable buf.h. inside mb_query.
       #mb_query.conf.buffer_handler := false;

       // Run the query.
       #mb_query(data_ptr := #dommy);

       #mb_query.conf.buffer_handler := true; // Enable buf.h. again.
       #mb_query.data_len := #mb_query.c.auto_len; // Back to auto.
   END_REGION

   REGION Insert & recive
       IF #mb_query.z.run.state = #INIT_QUERY  // Insert query.
           AND #mb_query.z.run.write
       THEN
           // Copy the content from data_ptr to the buffer.
           GATHER_BLK(IN := #data_ptr[#lower],
                      COUNT_OUT := #bytes,
                      OUT => #mb_query.z.buffer[0]);

       ELSIF  #mb_query.Done // The query above.
           AND NOT #mb_query.z.run.write  // A read query
       THEN
           // Copy the content from the buffer to data_ptr.
           SCATTER_BLK(IN := #mb_query.z.buffer[0],
                       COUNT_IN := #bytes,
                       OUT => #data_ptr[#lower]);
       END_IF;
   END_REGION
END_FUNCTION

FUNCTION "mb_execute" : Bool   // FC12, SCL
{ S7_Optimized_Access := 'TRUE' }
VERSION : 0.1
   VAR_IN_OUT
      mb_query : "mb_query";
   END_VAR
   VAR_TEMP
      dommy : Bool;
   END_VAR
BEGIN
   // Most use cases will not need this function !
   // Example:
   // 
   // IF "mb_execute"(#mb_query) THEN
   //     
   //     // Preparing calculations.
   //     
   //     #mb_query(data_addr := 2, data_ptr := #data);
   // END_IF;
   //
   // Usefull if some CPU demanding calculation need to be done
   // before a write query is inserted. Note that a query can later
   // be aborted, thought mb_execute return true.

   #mb_execute := #mb_query.z.run.qid_cnt + 1 = #mb_query.z.run.qid
   (* *)AND NOT #mb_query.stat.busy;

   IF NOT #mb_execute THEN
       #mb_query(data_ptr := #dommy);
   END_IF;
END_FUNCTION

// folder: Library/Modbus/Core/Special/Sequence

FUNCTION_BLOCK "mb_sequence"   // FB21, SCL
{ S7_Optimized_Access := 'TRUE' }
VERSION : 0.1
   VAR_IN_OUT
      sb : "mb_station_block_udt";   // Station block udt
      mb_query : "mb_query";
   END_VAR
   VAR
      Done : Bool;   // All queries has been exec. at least once, and no query has error.
      Error : Bool;   // At least one query has error.
      conf : Struct
         first_state : Int := 32767;   // Init state
      END_STRUCT;
      state : Int := 32767;
      next_state : Int := 32767;   // Will be transfer to state when query finnished
      z : Struct   // Internal variables
         first_scan : Bool := true;
         state_with_error : Int;
         a_query_is_executed : Bool;
      END_STRUCT;
   END_VAR
   VAR_TEMP
      write : Bool;
      exec : Bool;
   END_VAR
BEGIN
   // Controller for mb_query inside a state machine.

   // Figur out if the current state has a write query.
   CASE #mb_query.mode OF
       5, 6, 15, 16, 201, 202: // Write fc's.
           #write := true;
   END_CASE;

   // A query has executed, and there is a respons from device.
   #exec := #mb_query.Done
   (* *)OR #mb_query.Error AND NOT #mb_query.stat.error_comm;

   IF #sb.out.communication_error THEN
       IF #conf.first_state <> 32767 THEN
           #state := #conf.first_state;
       END_IF;
       #z.a_query_is_executed := #Done := false;

       // Go to next state, if the query in current state is a
       // write query and at the same time the read_only flag is set.
   ELSIF #exec OR #write AND #sb.conf.read_only THEN
       IF #exec THEN
           // Set the error flag, even when it's just one query in
           // the state machine that has an error.
           IF #mb_query.Error AND NOT #mb_query.stat.error_comm THEN
               #Error := true;
               #z.state_with_error := #state;
           ELSIF #mb_query.Done
               AND #z.state_with_error = #state
           THEN
               #Error := false;
           END_IF;

           // All queries has been executed at least once.
           IF #z.a_query_is_executed
               AND #state = #conf.first_state
               AND NOT #Error // No query with error.
           THEN
               #Done := true;
           END_IF;
           #z.a_query_is_executed := true;
       END_IF;

       // Change state
       #state := SEL(G := #next_state = 32767,
                     IN0 := #next_state,
                     IN1 := #state + 1);
   ELSE
       #mb_query.z.sb.seq_release := false;
   END_IF;

   IF #Error THEN
       #sb.z.err_hold := #sb.out.error := true;
   END_IF;

   #next_state := 32767;
   #z.first_scan := false;
END_FUNCTION_BLOCK

FUNCTION "mb_sequence_init" : Int   // FC7, SCL
{ S7_Optimized_Access := 'TRUE' }
VERSION : 0.1
   VAR_IN_OUT
      sequence : "mb_sequence";
      mb_query : "mb_query";
   END_VAR
BEGIN
   #mb_query.Done := #mb_query.Error := false;
   #mb_query.mode := INT_TO_USINT(#sequence.state / 100);

   IF #sequence.z.first_scan 
       AND #sequence.conf.first_state <> 32767
   THEN
       #sequence.state := #sequence.conf.first_state;
   END_IF;

   #mb_sequence_init := #sequence.state;
END_FUNCTION

// folder: Library/Modbus/Core/Special/Special code snippets examples

FUNCTION_BLOCK "Example Done and error"   // FB56, SCL
{ S7_Optimized_Access := 'TRUE' }
VERSION : 0.1
   VAR_IN_OUT
      mb_query : "mb_query";
   END_VAR
   VAR
      query1_data : Word;
      done_cnt : UInt;
      query2_data : Word;
   END_VAR
BEGIN
   // To get information about when a particular query has executed.

   #mb_query(mb_addr := 123,
             mode := #mb_query.c.write.holding_reg,
             data_addr := 456,
             data_ptr := #query1_data);

   // The if-statement bellow has to be put after the particular 
   // query, and before the next query.    

   IF #mb_query.Done THEN
       // Some action after a successfully query.    
       #done_cnt += 1; // Eg. count successfully queries.

   ELSIF #mb_query.Error THEN
       // Some action if a faild query.    

       // #mb_query.stat.status , gives more information about 
       // the error.         

       IF #mb_query.stat.error_comm THEN
           ; // Some particular action if communication error.
       END_IF;

   END_IF;

   // Next query...
   #mb_query(mb_addr := 111,
             mode := #mb_query.c.read.holding_reg,
             data_addr := 789,
             data_ptr := #query2_data);
END_FUNCTION_BLOCK

FUNCTION_BLOCK "Example Swap"   // FB78, SCL
{ S7_Optimized_Access := 'TRUE' }
VERSION : 0.1
   VAR_IN_OUT
      mb_query : "mb_query";
   END_VAR
   VAR
      static_tmp_var : Word;
      value : Word;
   END_VAR
BEGIN
   // For some modbus devices, when two registers are combined into one,
   // the data is stored as little endian, not big endian like Siemens 
   // PLC does. To solve this, the SWAP function needs to be utilized.
   #mb_query(mb_addr := 123,
             mode := #mb_query.c.read.holding_reg,
             data_addr := 123,
             data_ptr := #static_tmp_var);

   #value := SWAP(#static_tmp_var);


   // For other device, when two registers are combined, the least significant 
   // word is stored first and the most significant word is stored in the 
   // following register. When this is the case, the ROR-function needs 
   // to be used.
   #mb_query(mb_addr := 123,
             mode := #mb_query.c.read.holding_reg,
             data_addr := 123,
             data_ptr := #static_tmp_var);

   #value := ROR(IN := #static_tmp_var, N := 16);


   // In some situation both SWAP and ROR need to be used.
   #mb_query(mb_addr := 123,
             mode := #mb_query.c.read.holding_reg,
             data_addr := 123,
             data_ptr := #static_tmp_var);

   #value := SWAP(ROR(IN := #static_tmp_var, N := 16));

   // How the data is stored, is usually described in the
   // data sheet of each device.
END_FUNCTION_BLOCK

FUNCTION_BLOCK "Example Read first"   // FB85, SCL
{ S7_Optimized_Access := 'TRUE' }
VERSION : 0.1
   VAR_INPUT
      input1 : Bool;
      input2 : Bool;
   END_VAR
   VAR_IN_OUT
      mb_query : "mb_query";
   END_VAR
   VAR
      write : Bool;
      data : Word;
   END_VAR
BEGIN
   // Sometimes only some bits in a word need to be manipulated, 
   // without touching the other bits, bellow is an example how 
   // that can be achieved.

   #mb_query.mb_addr := 123;
   #mb_query.data_addr := 456;

   IF #write THEN // (Initially false)

       // Manipulating only bit 5 and 11
       #data.%X5 := #input1;
       #data.%X11 := #input2;

       #mb_query(mode := #mb_query.c.write.holding_reg,
                 data_ptr := #data);

   ELSE // read the register before write to the same one.
       #mb_query(mode := #mb_query.c.read.holding_reg,
                 data_ptr := #data);

       // Has query above been executed successfully?
       IF #mb_query.Done THEN
           #write := true;
       END_IF;

   END_IF;

   // Note: The read only option (#sb.conf.read_conly) can't be
   // used when the metod above is used.
END_FUNCTION_BLOCK

FUNCTION_BLOCK "Example Forced execution order"   // FB89, SCL
{ S7_Optimized_Access := 'TRUE' }
VERSION : 0.1
   VAR_IN_OUT
      mb_query : "mb_query";
   END_VAR
   VAR
      state : Int;
      query_1 : Word;
      query_2 : UInt;
      query_3 : Word;
      query_4 : Word;
   END_VAR
BEGIN
   // If the execution need to be forced to a given order, then the 
   // example bellow can be followed.

   CASE #state OF

       0:  // 1st query
           #mb_query(mb_addr := 123,
                     mode := #mb_query.c.write.holding_reg,
                     data_addr := 123,
                     data_ptr := #query_1);
           #state += BOOL_TO_SINT(#mb_query.Done);
           // «#mb_query.done» is set true when the query above is done 
           // successfully. When next query is executed, «#mb_query.done»
           // is set back false.

       1:  // 2nd query
           #mb_query(mb_addr := 123,
                     mode := #mb_query.c.write.holding_reg,
                     data_addr := 456,
                     data_ptr := #query_2);
           #state += BOOL_TO_SINT(#mb_query.Done);

       2:  // 3rd query
           #mb_query(mb_addr := 123,
                     mode := #mb_query.c.read.holding_reg,
                     data_addr := 789,
                     data_ptr := #query_3);
           IF #mb_query.Done THEN
               #state := 0;
           END_IF;

   END_CASE;

   // 4th query, this query is executed three times as often 
   // as the queries above.
   #mb_query(mb_addr := 123,
             mode := #mb_query.c.read.input_reg,
             data_addr := 1234,
             data_ptr := #query_4);


   // If the state machine has both read and write queries then
   // #sb.conf.read_only can't be used.
END_FUNCTION_BLOCK

FUNCTION_BLOCK "Example discrete queries"   // FB101, SCL
{ S7_Optimized_Access := 'TRUE' }
VERSION : 0.1
   VAR_IN_OUT
      mb_query : "mb_query";
   END_VAR
   VAR
      one_bool : Bool;
      two_bools : Struct
         b1 : Bool;
         b2 : Bool;
      END_STRUCT;
   END_VAR
BEGIN
   // Discrete queries.

   // When doing discrete queries the data_len parameter need to
   // be specified manualy.
   #mb_query(mb_addr := 123,
             mode := #mb_query.c.read.discrete_input,
             data_addr := 456,
             data_len := 1,
             data_ptr := #one_bool); // A single boolean.

   // Another quering two bool's
   #mb_query(mb_addr := 123,
             mode := #mb_query.c.read.discrete_input,
             data_addr := 789,
             data_len := 2,
             data_ptr := #two_bools); // A struct with two boolean inside.

   // After discrete queries, data_len should be set back in to auto.
   #mb_query.data_len := #mb_query.c.auto_len;
END_FUNCTION_BLOCK

FUNCTION_BLOCK "Example sequence"   // FB103, SCL
{ S7_Optimized_Access := 'TRUE' }
VERSION : 0.1
   VAR_INPUT
      mb_addr : USInt;
   END_VAR
   VAR_IN_OUT
      mb_query : "mb_query";
   END_VAR
   VAR
      sb : "mb_station_block_udt";
      sequence : "mb_sequence";
      read1 : Word;
      read2 : Word;
      read3 : Word;
      write1 : Word;
      write2 : Word;
      write3 : Word;
   END_VAR
BEGIN
   "mb_station_block_header"(sb := #sb, mb_query := #mb_query);
   #mb_query.mb_addr := #mb_addr;

   // High priority queries:
   #mb_query(mode := #mb_query.c.read.holding_reg,
             data_addr := 12345,
             data_ptr := #write3);

   IF #sequence.Done THEN
       #mb_query(mode := #mb_query.c.write.holding_reg,
                 data_addr := 54321,
                 data_ptr := #write3);
   END_IF;

   // Low priority queries:
   // Some queries that doesn't need to be run so often, the state
   // machines bellow make low priority queries be executed less often.
   #sequence.conf.first_state := 1600;
   CASE "mb_sequence_init"(sequence := #sequence, mb_query := #mb_query) OF
           // --------- Read holding reg queries (3xx) ---------
       300: #mb_query(data_addr := 123, data_ptr := #read1);
       301: #mb_query(data_addr := 456, data_ptr := #read2);
       302: #mb_query(data_addr := 789, data_ptr := #read3);

           #sequence.next_state := 1600;
           // --------- Write holding reg queries (16xx) ---------     
       1600: #mb_query(data_addr := 654, data_ptr := #write1);
       1601: #mb_query(data_addr := 321, data_ptr := #write2);
           #sequence.next_state := 300;
       ELSE
           #sequence.state += 1;
   END_CASE;
   #sequence(sb := #sb, mb_query := #mb_query);

   "mb_station_block_footer"(sb := #sb, mb_query := #mb_query);
END_FUNCTION_BLOCK

// folder: Library/Modbus/Core/sb

FUNCTION "mb_station_block_header" : Void   // FC10, SCL
{ S7_Optimized_Access := 'TRUE' }
VERSION : 1.0
   VAR_IN_OUT
      sb : "mb_station_block_udt";
      mb_query : "mb_query";
   END_VAR
   VAR CONSTANT
      ORIGIN : USInt := 0;
   END_VAR
BEGIN
   // Rexhip - Extended modbus library.
   // Read the top section of mb_query for more documentation.

   // Skip everything !
   IF #sb.conf.skip_code THEN
       RETURN;
   END_IF;

   #mb_query.data_len := 0; // Default is auto-length.
   #mb_query.conf.buffer_handler := true;

   // If device blocks are executeded in diffrent order, a wide wind
   // up effect will occur, (in same OB) this will prevent that.
   IF #mb_query.z.sb.reset THEN
       #sb.z.header_qid := #mb_query.z.run.qid_cnt + 1;
   END_IF;

   // Device id cnt. The first device has id "1". Increased in every
   // mb_device_header, reseted in mb_client_ctrl or mb_master_ctrl.
   #mb_query.z.sb.sid_cnt += 1;

   // mb_query set the same bellow variables to true, at insert or recive.
   // This informastion is later used at the footer.
   #mb_query.z.sb.head_insert := false;
   #mb_query.z.sb.head_recive := false;

   // Reset order, a variable that makes queries in a sb execute in order.
   // #mb_query.z.sb.order := false;

   // When #mb.mb.q.qid = #mb.mb.run.qid_cnt => "This" device has the
   // query-token !
   // - If the query-token points at this device header, or it point to a
   //   query in the previous device, that is surrounded by a if-statement
   //   and the statement is now false.
   // - A gid change can only be done if not "busy", this is to avoid a
   //   resualt from one query being intercepted by another
   IF #mb_query.z.run.qid > #mb_query.z.run.qid_cnt
       AND #mb_query.z.run.qid <= #sb.z.header_qid
       AND NOT #mb_query.stat.busy
   THEN
       // Reset.
       // Go back to the first state in mb_query. New query param. will
       // owerwrite old once.
       #mb_query.z.run.state := #ORIGIN;

       // At first the offset_qid points at the first query of this
       // device. When it has executed the offset will point at the
       // second query. When all queries has executed the offset will
       // be reset back to the first query. (footer) 
       #mb_query.z.run.qid :=
       (* *)#sb.z.header_qid + #sb.z.offset_qid;

       // Order is a variable that makes queries in sb execute in order.
       //    #mb_query.z.sb.order := true;
   END_IF;

   // - The code below is reduce the impact of setting a if-statement
   //   around queries, by setting the qid_cnt to a fixed value at this 
   //   point.
   // - mb_station_block_header will occupy one query-id.  
   #sb.z.header_qid :=
   MAX(IN1 := #mb_query.z.run.qid_cnt + 1,
       IN2 := #sb.z.header_qid);
   #mb_query.z.run.qid_cnt := #sb.z.header_qid;
END_FUNCTION

FUNCTION "mb_station_block_footer" : Void   // FC11, SCL
{ S7_Optimized_Access := 'TRUE' }
VERSION : 1.0
   VAR_IN_OUT
      sb : "mb_station_block_udt";
      mb_query : "mb_query";
   END_VAR
   VAR_TEMP
      "e" : Int;
      err : Bool;
   END_VAR
   VAR CONSTANT
      INSERT_QUERY : USInt := 1;
   END_VAR
BEGIN
   // Rexhip - Extended modbus library.
   // Read the top section of mb_query for more documentation.

   // Skip everything !
   IF #sb.conf.skip_code THEN
       RETURN;
   END_IF;

   REGION Recive
       IF #mb_query.z.sb.head_recive THEN
           // If there is a query that bellong to this device that has
           // recvied a resault. (with or without error)

           // Counter for exec. queries inside this station block.
           // Default is 1 query for each loop, but may be changed.
           #sb.z.exec_cnt += 1;

           // If this is the first succesfylly query after communication error,
           // then log the time this happen. (also exceptions)
           IF #sb.out.communication_error AND (
               #mb_query.stat.done
               OR #mb_query.stat.error AND NOT #mb_query.stat.error_comm)
           THEN
               #"e" := RD_LOC_T(#sb.log.connected_time);
           END_IF;

           IF #mb_query.stat.error THEN // Logging - failed query        
               // Store the values for debugging. data_addr will indicate witch 
               // query caused the error, and the status is indicate the error type.
               #sb.log.error_status := #mb_query.stat.status;
               #sb.log.error_data_addr := #mb_query.z.sb.log_data_addr;

               // Two counters, one for comm.error and for all other errors.
               IF #mb_query.stat.error_comm THEN
                   #sb.log.error_comm_cnt += 1; // Eg. Bad CRC, parity, etc.
               ELSE
                   #sb.log.error_exception_cnt += 1;
               END_IF;

               // Increase communication error counter. if it's a comm.error.
               // then reset the counter.  
               IF #mb_query.stat.error_comm THEN
                   #sb.z.comm_err_cnt += BOOL_TO_USINT(#sb.z.comm_err_cnt < 255);
               ELSE
                   #sb.z.comm_err_cnt := 0;
               END_IF;

               // The error_comm flag is set if x repeating comm.errors occurres.
               #err := #sb.z.comm_err_cnt > #sb.conf.max_comm_error;
               IF #err AND NOT #sb.out.communication_error THEN
                   // Log the time when the flag is set.
                   #"e" := RD_LOC_T(#sb.log.disconnected_time);
               END_IF;
               #sb.out.communication_error := #err;

               // A comm.error will not be displayed before the
               // communication_error flag is set. Other errors will be
               // diplayed once. (NOT comm.error -> normal error)
               #sb.out.error := #sb.out.error OR NOT #mb_query.stat.error_comm
               OR #sb.out.communication_error;

               // err_hold makes the error flag stay true for more then just
               // one plc-scan.
               #sb.z.err_hold := #sb.out.error;

           ELSIF #mb_query.stat.done THEN // Logging successfully query        
               #sb.log.done_cnt += 1;
               // One successfully query -> reset fault.
               #sb.out.communication_error := false;
               #sb.z.comm_err_cnt := 0;
           END_IF;

           // - If it's this devices has the retry token, (sid_retry = sid_cnt)
           //   a retry has been executed and faild. Then set the retry_finished
           //   flag.
           // - The retry-token will be passed on to the next device with
           //   communication problems when the query loop has reach
           //   the end. (Inside the mb_internal_e)
           // - The library make sure that only one station block with comm.
           //   problems will do retry for each query loop revolution. 
           #mb_query.z.sb.sid_retry_finished :=
           #mb_query.z.sb.sid_retry = #mb_query.z.sb.sid_cnt
           AND #mb_query.stat.error_comm;

           // Only one query in the SB is executed (default). The purpose is
           // to avoid a SB with many queries to occupy the bus for long periodes
           // of time. offset_qid is incread by one when a query has executed
           // given last query didn't resualt in a timeout.
           #sb.z.offset_qid += BOOL_TO_UINT(NOT #mb_query.stat.error_comm);
       END_IF;
   END_REGION

   REGION Middle
       // If all queries for this device has been executed,
       // then reset offset_qid back to the first query.
       IF #sb.z.offset_qid >
           #mb_query.z.run.qid_cnt - #sb.z.header_qid
       THEN
           #sb.z.offset_qid := 1;

           // Also reset error falg, if the last query was successfully.
           IF NOT #sb.z.err_hold THEN
               #sb.out.error := false;
           END_IF;
           #sb.z.err_hold := false;
       END_IF;

       // If the retry-token point at this device (sid_retry=sid_cnt), and there is
       // no communication problems then pass on the retry-token to the next device.
       // The retry token tell which device with communication problem that should
       // retry establish communication.
       #mb_query.z.sb.sid_retry +=
       BOOL_TO_UINT(#mb_query.z.sb.sid_retry = #mb_query.z.sb.sid_cnt
                    AND NOT #sb.out.communication_error);
   END_REGION

   REGION Finnish
       // Several condition that resault in passing on the query-token on to the
       // next device. Skipping all or the rest of the queries for this device:              
       #sb.out.finnish :=
       #mb_query.z.sb.head_recive AND ( // Skip rest of the queries if: ->
       (* *)#sb.z.exec_cnt >= #sb.conf.exec_x_quries // Some queries has executed,
       (*           *)// wait for the next loop for the remaining queries.
       (*      *)OR #mb_query.stat.error_comm) // A query resualting in comm.error    
       OR #mb_query.z.sb.head_insert AND ( // Erase a already inserted query if: ->
       (* *)#sb.out.communication_error // This station has allready comm. problems.
       (*      *)// And, it isn't this devies turn to try again.
       (*      *)AND (#mb_query.z.sb.sid_retry <> #mb_query.z.sb.sid_cnt
       (*           *)// Or, there has allready been a retry attempt on this loop.
       (*           *)OR #mb_query.z.sb.sid_retry_finished) // (reseted in mb_internal_e)     
       (* *)OR #sb.conf.disable    
       (* *)OR #sb.conf.exec_x_quries = 0 // Zero => disable station block.
       (* *)OR #sb.conf.read_only // The read_only flag is set, and it's a write query.
       (*      *)AND #mb_query.z.run.write);

       IF #sb.out.finnish THEN // Reset
           // Go back to the first state in mb_query. New query param. will owerwrite 
           // old once.
           #mb_query.z.run.state := #INSERT_QUERY;
           // Set to qid to the next station block.
           #mb_query.z.run.qid := #mb_query.z.run.qid_cnt + 1;
           #sb.z.exec_cnt := 0;

           // If the sb is read only mode and a write query is hit, then skip it
           // and advance to the next query on the next run.
           #sb.z.offset_qid +=
           (* *)BOOL_TO_UINT(#sb.conf.read_only AND #mb_query.z.run.write);        
       END_IF;
   END_REGION
END_FUNCTION

// folder: Library/Modbus/Core/z Internal

FUNCTION_BLOCK "mb_internal_b"   // FB6, SCL
{ S7_Optimized_Access := 'FALSE' }
VERSION : 0.1
   VAR
      buffer : Array[0..249] of Byte;
   END_VAR
BEGIN
   (*
   - Buffer for mb_master and modbus_master. (modbus rtu)
   - This block has optimize data access disabled.
   - For RTU, please do not delete the even there is no code bellow.
   - This block isn't needed for modbus tcp.
   *)
END_FUNCTION_BLOCK

FUNCTION_BLOCK "mb_internal_e"   // FB7, SCL
{ S7_Optimized_Access := 'TRUE' }
VERSION : 0.1
   VAR_OUTPUT
      Error : Bool;
   END_VAR
   VAR_IN_OUT
      mb_query : "mb_query";
   END_VAR
   VAR
      err_hold : Bool;
   END_VAR
   VAR CONSTANT
      INSERT_QUERY : USInt := 1;
      EXEC_QUERY : USInt := 3;
      RECIVE_RESUALT : USInt := 4;
   END_VAR
BEGIN
   // Internal function - common for both rtu and tcp.

   // Move on to next state when query is finnished.
   IF #mb_query.z.run.state = #EXEC_QUERY 
       AND (#mb_query.stat.error OR #mb_query.stat.done)
   THEN
       #mb_query.z.run.state := #RECIVE_RESUALT;
   END_IF;


   // Anti wind up effect for qid. msg. to devices that they should
   // reset if qid grow bigger then 60000. (See mb_station_block_header)
   #mb_query.z.sb.reset := false;
   IF #mb_query.z.run.qid > 60000 THEN
       #mb_query.z.sb.reset := true;
   END_IF;

   // #error will be keeped true as long there is at least one query that
   // generate a error. 
   IF #mb_query.stat.error THEN
       #Error := true;
       #err_hold := true;
   END_IF;

   // If all queries has been executed,
   IF #mb_query.z.run.qid > #mb_query.z.run.qid_cnt THEN

       // Error handeling (see above)
       IF NOT #err_hold THEN
           #Error := false;
       END_IF;
       #err_hold := false;

       // Start over again on the first query.
       #mb_query.z.run.qid := 1;

       // The retry-id is the device that get to have retry to restoring
       // communication after the error_comm flag is set for the station.
       // When one query loop has occurred the retry id is incremented. 
       #mb_query.z.sb.sid_retry := #mb_query.z.sb.sid_retry + 1;

       // retry_finished is set after one retry has taken place. 
       // The station that has the retry-token only has one try to make 
       // successfully query.
       #mb_query.z.sb.sid_retry_finished := false;
       IF #mb_query.z.sb.sid_retry > #mb_query.z.sb.sid_cnt THEN
           #mb_query.z.sb.sid_retry := 1;
       END_IF;

       // Station id (sid):
       // A sb can do some action, when sid_cnt is equal it's sid.
       // If sid_halt is set true, sid inc. will then stop until it's
       // released. 
       #mb_query.z.sb.sid := #mb_query.z.sb.sid
       (* *)+ BOOL_TO_UINT(NOT #mb_query.z.sb.sid_halt);
       #mb_query.z.sb.sid_halt := false;
       IF #mb_query.z.sb.sid > #mb_query.z.sb.sid_cnt THEN
           #mb_query.z.sb.sid := 1;
       END_IF;
   END_IF;

   #mb_query.z.run.qid_cnt := 0; // (Incremented in mb_query)
   #mb_query.z.sb.sid_cnt := 0; // (Incremented in mb_station_block_header)
END_FUNCTION_BLOCK

FUNCTION "mb_internal_f" : Void   // FC2, SCL
{ S7_Optimized_Access := 'TRUE' }
VERSION : 0.1
   VAR_IN_OUT
      buffer : "mb_internal_b";
      mb_query : "mb_query";
   END_VAR
   VAR_TEMP
      comm_error : Bool;
   END_VAR
BEGIN
   // Internal function - master footer

   IF #mb_query.stat.error THEN
       // Figur out if it's a communication error.
       // (Handled different from other errors)
       CASE WORD_TO_UINT(#mb_query.stat.status) OF
           16#80C8, // Timeout
           16#80E1, // Parity error
           16#80E2, // Framing error
           16#8380: // Bad CRC 
               #comm_error := true;
       END_CASE;

   ELSIF #mb_query.stat.done // Successful query
       AND NOT #mb_query.z.run.write // A read query.
   THEN
       #mb_query.z.buffer := #buffer.buffer;
   END_IF;

   #mb_query.stat.error_comm :=
   (* *)#mb_query.stat.error AND #comm_error;
END_FUNCTION

FUNCTION "mb_internal_a" : Void   // FC4, SCL
{ S7_Optimized_Access := 'TRUE' }
VERSION : 0.1
   VAR_INPUT
      mode104 : Bool;
   END_VAR
   VAR_OUTPUT
      Mode : USInt;
      Data_addr : UDInt;
   END_VAR
   VAR_IN_OUT
      mb_query : "mb_query";
   END_VAR
BEGIN
   // Internal function

   // Modicon convention address.
   #Mode := 0;
   CASE #mb_query.z.q.mode OF
       1:  // Read output bits
           #Data_addr := 1 + #mb_query.z.q.data_addr;
       2:  // Read input bits
           #Data_addr := 10001 + #mb_query.z.q.data_addr;
       3:  // Read holding reg.
           #Data_addr := 400001 + #mb_query.z.q.data_addr;
       4:  // Read input word
           IF #mode104 THEN
               #Mode := 104;
               #Data_addr := #mb_query.z.q.data_addr;
           ELSE
               #Data_addr := 30001 + #mb_query.z.q.data_addr;
           END_IF;
       5:  // Writing a single output bit
           #Mode := 1;
           #Data_addr := 1 + #mb_query.z.q.data_addr;
       6:  // Writing a single holding register
           #Mode := 1;
           #Data_addr := 400001 + #mb_query.z.q.data_addr;
       15: // Writing multiple output bits
           #Mode := 2;
           #Data_addr := 1 + #mb_query.z.q.data_addr;
       16: // Writing multiple holding registers
           #Mode := 2;
           #Data_addr := 400001 + #mb_query.z.q.data_addr;
       200..202: // Read and write
           #Mode := #mb_query.z.q.mode - 200;
           #Data_addr := #mb_query.z.q.data_addr;
       ELSE
           #Mode := #mb_query.z.q.mode;
           #Data_addr := #mb_query.z.q.data_addr;
   END_CASE;
END_FUNCTION

FUNCTION "mb_timeout_rtu_calc" : Time   // FC5, SCL
{ S7_Optimized_Access := 'TRUE' }
VERSION : 0.1
   VAR_INPUT
      gain : Real;
      offset : Time;
      baud : UDInt;
   END_VAR
   VAR_IN_OUT
      mb_query : "mb_query";
   END_VAR
   VAR_TEMP
      t : Time;
   END_VAR
BEGIN
   // Automatically adjust timeout for modbus rtu.

   IF #gain = 0 THEN
       #t := #offset;
   ELSE
       #t := T_CONV
       (REAL_TO_UINT
        (
         11000 * ( //  11: Bits: start, data, parity, stop. 
         (* *)//   * 1000: Seconds to milliseconds
         (* *)19 // Bytes: Req: mb_addr, fc, data_addr(2), data_len(2), crc(2), 
         (* *) //        + res: mb_addr, fc, byte-count, crc(2), 
         (* *) //        + start-stop -> 6 (ca 2 x 28 bits)
         (* *)+ UINT_TO_REAL(#mb_query.z.q.data_len) *
         (*     *)SEL(G := #mb_query.z.run.discrete,
                      (* *)IN0 := INT_TO_REAL(2), // Each word is to bytes.
                      (* *)IN1 := 0.125) // Eight bits in one byte. (1/8 = 0.125)
         )
         / UDINT_TO_REAL(#baud) // High baud-rate -> low timeout
         * #gain // Safty margin
         + UDINT_TO_UINT(T_CONV(#offset))
        ));
   END_IF;

   #mb_timeout_rtu_calc :=
   LIMIT(MN := T#5ms, // A least 5ms, else comm_load will throw a error.
         IN := #t,
         MX := T#65s);
END_FUNCTION

// folder: Library/Modbus/Core/z Testing

FUNCTION_BLOCK "rtu_test1_1200"   // FB3, SCL
{ S7_Optimized_Access := 'TRUE' }
VERSION : 0.1
   VAR
      mb_query : "mb_query";
      mb_master_1200_ctrl : "mb_master_1200_ctrl";
      delay_between_queries : "mb_delay_between_queries";
      delay : "mb_delay";
      __ : Bool;
      temperature_1 : "Jdrk_RS_WS_N01_8";
      temperature_2 : "Jdrk_RS_WS_N01_8";
      temperature_3 : "Jdrk_RS_WS_N01_8";
      sb_temp_no_answer_1 : "sb_temp_no_answer";
      sb_temp_no_answer_2 : "sb_temp_no_answer";
      sb_temp_no_answer_3 : "sb_temp_no_answer";
      sb_temp_error_1 : "sb_temp_error";
      sb_temp_error_2 : "sb_temp_error";
      sb_temp_error_3 : "sb_temp_error";
      _ : Bool;
      bool_arrary : Array[0..15] of Bool;
      sb : "mb_station_block_udt";
   END_VAR
BEGIN
   #mb_master_1200_ctrl.conf.parity := 0;
   #mb_master_1200_ctrl(hardware_id := 269, // "Local~CB_1241_(RS485)",
                        baud := 9600,
                        mb_query := #mb_query);

   #delay_between_queries(mb_query := #mb_query);

   #temperature_1(mb_query := #mb_query);
   #temperature_2(mb_query := #mb_query);
   #temperature_3(mb_query := #mb_query);

   #delay(mb_query := #mb_query);

   #sb_temp_no_answer_1(mb_query := #mb_query);
   #sb_temp_no_answer_2(mb_query := #mb_query);
   #sb_temp_no_answer_3(mb_query := #mb_query);

   #sb_temp_error_1(mb_query := #mb_query);
   #sb_temp_error_2(mb_query := #mb_query);
   #sb_temp_error_3(mb_query := #mb_query);

   "mb_station_block_header"(sb := #sb, mb_query := #mb_query);
   #mb_query.mb_addr := 1;
   #mb_query.mode := #mb_query.c.read.input_reg;
   #mb_query.data_addr := 1;
   "mb_query_bits"(data_ptr := #bool_arrary, mb_query := #mb_query);
   "mb_station_block_footer"(sb := #sb, mb_query := #mb_query);
END_FUNCTION_BLOCK

FUNCTION_BLOCK "tcp_test"   // FB96, SCL
{ S7_Optimized_Access := 'TRUE' }
VERSION : 0.1
   VAR
      mb_query : "mb_query";
      mb_client_ctrl : "mb_client_ctrl";
      t1 : Word;
      t2 : Word;
      t3 : Word;
      t4 : Word;
      aa : Bool;
      mb_delay_between_queries : "mb_delay_between_queries";
      sb : "mb_station_block_udt";
   END_VAR
BEGIN

   #mb_client_ctrl.ip_addr[1] := 192;
   #mb_client_ctrl.ip_addr[2] := 168;
   #mb_client_ctrl.ip_addr[3] := 0;
   #mb_client_ctrl.ip_addr[4] := 33;
   #mb_client_ctrl(interface := 64,
                   conn_id := 123,
                   tcp_port := 502,
                   // timeout := T#500ms,
                   mb_query := #mb_query);

   #mb_delay_between_queries(// delay := T#1s,
                             mb_query := #mb_query);

   "mb_station_block_header"(sb := #sb, mb_query := #mb_query);

   #mb_query(mb_addr := 255,
             mode := #mb_query.c.write.holding_reg,
             data_addr := 1,
             data_ptr := #t1);

   #mb_query(mode := #mb_query.c.read.holding_reg,
             data_addr := 1,
             data_ptr := #t2);

   #mb_query(mode := #mb_query.c.write.holding_reg,
             data_addr := 2,
             data_ptr := #t2);

   #mb_query(mode := #mb_query.c.read.holding_reg,
             data_addr := 2,
             data_ptr := #t3);

   "mb_station_block_footer"(sb := #sb, mb_query := #mb_query);
END_FUNCTION_BLOCK

FUNCTION_BLOCK "rtu_test2_1200"   // FB98, SCL
{ S7_Optimized_Access := 'TRUE' }
VERSION : 0.1
   VAR
      mb_query : "mb_query";
      mb_master_1200_ctrl : "mb_master_1200_ctrl";
      Danfoss : "Danfoss_VLT";
      Mjk_expert_1 : "Mjk_expert";
      Mjk_expert_2 : "Mjk_expert";
      Mjk_expert_3 : "Mjk_expert";
   END_VAR
BEGIN
   #mb_master_1200_ctrl.conf.parity := 0;
   #mb_master_1200_ctrl(hardware_id := 0, // "Local~CB_1241_(RS485)",
                        baud := 9600,
                        mb_query := #mb_query);

   #Mjk_expert_1(mb_addr := 1, mb_query := #mb_query);
   #Mjk_expert_2(mb_addr := 1, mb_query := #mb_query);
   #Mjk_expert_3(mb_addr := 1, mb_query := #mb_query);

   #Danfoss(mb_addr := 2, mb_query := #mb_query);
END_FUNCTION_BLOCK

FUNCTION_BLOCK "rtu_test_1500"   // FB102, SCL
{ S7_Optimized_Access := 'TRUE' }
VERSION : 0.1
   VAR
      mb_master_1500_ctrl : "mb_master_1500_ctrl";
      mb_query : "mb_query";
      temperature_1 : "Jdrk_RS_WS_N01_8";
      temperature_2 : "Jdrk_RS_WS_N01_8";
      temperature_3 : "Jdrk_RS_WS_N01_8";
      sb_temp_no_answer_1 : "sb_temp_no_answer";
      sb_temp_no_answer_2 : "sb_temp_no_answer";
      sb_temp_no_answer_3 : "sb_temp_no_answer";
      sb_temp_error_1 : "sb_temp_error";
      sb_temp_error_2 : "sb_temp_error";
      sb_temp_error_3 : "sb_temp_error";
      delay_between_queries : "mb_delay_between_queries";
      mb_delay : "mb_delay";
   END_VAR
BEGIN

   #mb_master_1500_ctrl.conf.parity := 0;
   #mb_master_1500_ctrl(hardware_id := 269,
                        operating_mode := 4,
                        baud := 9600,
                        mb_query := #mb_query);

   #delay_between_queries(mb_query := #mb_query);


   #temperature_1(mb_query := #mb_query);
   #temperature_2(mb_query := #mb_query);
   #temperature_3(mb_query := #mb_query);

   #mb_delay(mb_query := #mb_query);

   #sb_temp_no_answer_1(mb_query := #mb_query);
   #sb_temp_no_answer_2(mb_query := #mb_query);
   #sb_temp_no_answer_3(mb_query := #mb_query);

   #sb_temp_error_1(mb_query := #mb_query);
   #sb_temp_error_2(mb_query := #mb_query);
   #sb_temp_error_3(mb_query := #mb_query);
END_FUNCTION_BLOCK

// folder: Library/Modbus/Core/z Testing/sb

FUNCTION_BLOCK "sb_temp_no_answer"   // FB32, SCL
{ S7_Optimized_Access := 'TRUE' }
VERSION : 0.1
   VAR_OUTPUT
      Temperature : Real;
   END_VAR
   VAR_IN_OUT
      mb_query : "mb_query";
   END_VAR
   VAR
      sb : "mb_station_block_udt";
   END_VAR
   VAR RETAIN
      offset : Real;
   END_VAR
   VAR_TEMP
      tmp : Int;
   END_VAR
BEGIN
   // JDRK - RS-WS-N01-8 - Temperature and Humidity sensor

   "mb_station_block_header"(sb := #sb, mb_query := #mb_query);

   #mb_query(mb_addr := 200,
             mode := #mb_query.c.read.input_reg,
             data_addr := 1,
             data_ptr := #tmp);

   IF #mb_query.Done THEN
       #Temperature := INT_TO_REAL(#tmp) / 10 + #offset;
   END_IF;

   "mb_station_block_footer"(sb := #sb, mb_query := #mb_query);
END_FUNCTION_BLOCK

FUNCTION_BLOCK "sb_temp_error"   // FB33, SCL
{ S7_Optimized_Access := 'TRUE' }
VERSION : 0.1
   VAR_OUTPUT
      Temperature : Real;
   END_VAR
   VAR_IN_OUT
      mb_query : "mb_query";
   END_VAR
   VAR
      sb : "mb_station_block_udt";
   END_VAR
   VAR RETAIN
      tt : Array[0..100] of Int;
   END_VAR
   VAR_TEMP
      tmp : Int;
   END_VAR
BEGIN
   // JDRK - RS-WS-N01-8 - Temperature and Humidity sensor

   "mb_station_block_header"(sb := #sb, mb_query := #mb_query);

   #mb_query(mb_addr := 1,
             mode := #mb_query.c.read.input_reg,
             data_addr := 1,
             data_ptr := #tmp);

   IF #mb_query.Done THEN
       #Temperature := INT_TO_REAL(#tmp) / 10;
   END_IF;

   // Query producing a error.
   #mb_query(mb_addr := 1,
             mode := #mb_query.c.read.input_reg,
             data_addr := 1,
             data_ptr := #tt);

   "mb_station_block_footer"(sb := #sb, mb_query := #mb_query);
END_FUNCTION_BLOCK

// folder: Library/Modbus/Docs

FUNCTION "mb_Debugging" : Void   // FC1, SCL
{ S7_Optimized_Access := 'TRUE' }
VERSION : 0.1
BEGIN
   (* 
   # General debugging:
   - Look online and check that the latest version of the library 
     is in use.
   - All queries need to be executed in same order, implicates from 
     the same OB.
   - Look inside the data blcok of the SB of the device that having 
     problem, and locate «#sb.log...», see if the counters are 
     running and lookup the error code of «#sb.log.error_status», 
     «#sb.log.error_data_addr» will tell witch query generating the 
     error. 

   # Modbus RTU
   - Try to increase timeout, repeaters on the bus need additional 
     time.
   - All the devies on the bus need to have a unique address.
   - Parity, buard rate, stop bits need to be the same in all 
     devices. The modbus specification state on page 20, that 19200
     is the default/recommended buad rate. The specification also 
     state, on page 12, that parity should be "even".
   - Electrical polarity, for some devices the connection "A" and "B" 
     is mislabeled, try to swap them.
   - Check for correct hardware id,

   # Modbus TCP
   - Try to increase timeout, creating a TCP-socket may take long.
   - Check IP-address.
   - Check TCP-port, 502 is default.
   - Check for unic connection-id.

   # Station Blocks 
   - If mb_station_block_header has executed in one block then 
     mb_station_block_foother also need to be executed. Cheack that 
     there is no RETURN or simular between them.
   - Check datasheet of device for special requirement: function codes 
     supported, max data length, register required to be queried 
     together, etc.  
   - A query can't be longer then 124 words.   
   - Try to comment out queries and see if it solve the problem.  

   *)
END_FUNCTION

// folder: Library/Modbus/Station blocks/sb tested

FUNCTION_BLOCK "Mjk_expert"   // FB35, SCL
{ S7_Optimized_Access := 'TRUE' }
VERSION : 0.1
   VAR_INPUT
      mb_addr : USInt;
   END_VAR
   VAR_IN_OUT
      mb_query : "mb_query";
   END_VAR
   VAR
      sb : "mb_station_block_udt";
      data : Struct
         pressure : Real;
         temperature : Real;
      END_STRUCT;
   END_VAR
BEGIN
   // MJK - Expert 700-7060-7070 - Pressure transmitters

   "mb_station_block_header"(sb := #sb, mb_query := #mb_query);
   #mb_query.mb_addr := #mb_addr;

   #mb_query.mode := #mb_query.c.read.holding_reg;
   #mb_query(data_addr := 16#100, data_ptr := #data);

   "mb_station_block_footer"(sb := #sb, mb_query := #mb_query);

   (*
       Rød     +24V
       Brown   GND
       Yellow  RS485 B
       Gray    RS485 A
       White   Voltage output
   *)
END_FUNCTION_BLOCK

// folder: Library/Modbus/Station blocks/sb tested/Danfoss

FUNCTION_BLOCK "Danfoss_VLT"   // FB71, SCL
{ S7_Optimized_Access := 'TRUE' }
VERSION : 0.1
   VAR_INPUT
      mb_addr : USInt;
      iRef : Real;   // [%]
      iCost : Bool;
      iDC_break : Bool;
      iStop_quick : Bool;
      iReset : Bool;
   END_VAR
   VAR_OUTPUT
      qReady : Bool;
      qRunning : Bool;
      qError : Bool;
      qIn_operation : Bool;
      qIn_auto : Bool;
      qPower : Real;   // [kw]
      qCurrent : Real;   // [A]
      qFreq_hz : Real;   // [hz]
      qSpeed_rpm : Real;   // [rpm]
      qVoltage : Real;
      qOutput_percent : Real;
      qTorque_percent : Int;
      qHeatsink_temp : Int;
      qAlarm_word : DWord;
   END_VAR
   VAR_IN_OUT
      mb_query : "mb_query";
   END_VAR
   VAR
      sb : "mb_station_block_udt";
   END_VAR
   VAR RETAIN
      conf : Struct
         Send_config_to_drive : Bool := true;
         action_no_communication : Int := 2;   // 2: Stop,
         input_source : Int := 2;   // 2: ctw fieldbus
      END_STRUCT;
   END_VAR
   VAR
      read : Struct   // (unscaled)
         stw : Struct   // Status word
            speed_eq_reference : Bool;   // [08]
            bus_control : Bool;   // [09] false=hand mode
            frequency_limit_ok : Bool;   // [10]
            in_operation : Bool;   // [11]
            stopped_auto_start : Bool;   // [12]
            voltage_exceeded : Bool;   // [13]
            torque_exceeded : Bool;   // [14]
            timer_exceeded : Bool;   // [15]
            control_ready : Bool;   // [00]
            drive_ready : Bool;   // [01]
            enable : Bool;   // [02] 0=Coasting
            trip : Bool;   // [03]
            error_no_trip : Bool;   // [04]
            x05 : Bool;   // [05]
            triplock : Bool;   // [06]
            warning : Bool;   // [07]
         END_STRUCT;
         man : Int;   // man actual value
      END_STRUCT;
      write : Struct   // Controll word
         ctw : Struct   // Controll word
            x08 : Bool;   // [08]
            use_ramp_2 : Bool;   // [09]
            data_valid : Bool := TRUE;   // [10]
            x11 : Bool;   // [11]
            x12 : Bool;   // [12]
            x13 : Bool;   // [13]
            x14 : Bool;   // [14]
            reverse : Bool;   // [15]
            x00 : Bool;   // [00]
            x01 : Bool;   // [01]
            dc_break_NOT : Bool := TRUE;   // [02]
            coast_NOT : Bool := TRUE;   // [03]
            quick_stop_NOT : Bool := TRUE;   // [04]
            hold_output_frequency_NOT : Bool := TRUE;   // [05]
            start : Bool;   // [06]
            reset : Bool;   // [07]
         END_STRUCT;
         ref : Int;
      END_STRUCT;
      sequence : "mb_sequence";
   END_VAR
   VAR_TEMP
      tmp : Int;
      dtmp : DInt;
   END_VAR
BEGIN
   (* Danfoss - VLT

       doc_MG20N202.pdf
       doc_MG20O602.pdf 
   *)

   "mb_station_block_header"(sb := #sb, mb_query := #mb_query);
   #mb_query.mb_addr := #mb_addr;

   REGION Low priority queries
       // Some queries that doesn't need to be run so often, the state
       // machines bellow make low priority queries be executed less often. 
       #sequence.conf.first_state := SEL(G := #conf.Send_config_to_drive
                                         AND NOT #sb.conf.read_only,
                                         IN0 := 300, IN1 := 1600);

       CASE "mb_sequence_init"(sequence := #sequence, mb_query := #mb_query) OF

               // --------- Read holding reg queries ---------

           300:  // Freq hz 
               #mb_query(data_addr := "p"(a := 16, b := 13), data_ptr := #tmp);
               IF #mb_query.Done THEN
                   #qFreq_hz := DINT_TO_REAL(#tmp) * 0.1;
               END_IF;
           301:  // Electrical current 
               #mb_query(data_addr := "p"(a := 16, b := 14), data_ptr := #dtmp);
               IF #mb_query.Done THEN
                   #qCurrent := DINT_TO_REAL(#dtmp) * 0.01;
               END_IF;
           302:  // RPM
               #mb_query(data_addr := "p"(a := 16, b := 17), data_ptr := #dtmp);
               IF #mb_query.Done THEN
                   #qSpeed_rpm := DINT_TO_REAL(#dtmp) / 60;
               END_IF;
           303:  // Power
               #mb_query(data_addr := "p"(a := 16, b := 10), data_ptr := #dtmp);
               IF #mb_query.Done THEN
                   #qPower := DINT_TO_REAL(#dtmp) * 10;
               END_IF;
           304:  // Heatsink Temp. 
               #mb_query(data_addr := "p"(a := 16, b := 34), data_ptr := #tmp);
               IF #mb_query.Done THEN
                   #qHeatsink_temp := #tmp;
               END_IF;
           305:  // Motor voltage
               #mb_query(data_addr := "p"(a := 16, b := 12), data_ptr := #tmp);
               IF #mb_query.Done THEN
                   #qVoltage := INT_TO_REAL(#tmp) * 0.1;
               END_IF;
           306:  // Alarm word 
               #mb_query(data_addr := "p"(a := 16, b := 92), data_ptr := #dtmp);
               IF #mb_query.Done THEN
                   #qAlarm_word := DINT_TO_DWORD(#dtmp);
               END_IF;
           307:  // Torque [%] 
               #mb_query(data_addr := "p"(a := 16, b := 22), data_ptr := #tmp);
               IF #mb_query.Done THEN
                   #qTorque_percent := #tmp;
               END_IF;

               #sequence.next_state := #sequence.conf.first_state;

               // --------- Write holding reg queries ---------     

           1600: // Action if no communication. (2=stop)     
               #mb_query(data_addr := "p"(a := 8, b := 4),
                         data_ptr := #conf.action_no_communication);
           1601: // Select input source (2=CTW=fieldbus)     
               #mb_query(data_addr := "p"(a := 8, b := 1),
                         data_ptr := #conf.input_source);

               #sequence.next_state := 300;
           ELSE
               #sequence.state += 1;
       END_CASE;
       #sequence(sb := #sb, mb_query := #mb_query);
   END_REGION

   REGION High priority queries
       // Status word  and main actual value 
       #mb_query(mode := #mb_query.c.read.holding_reg,
                 data_addr := 2909,
                 data_ptr := #read);
       IF #mb_query.Done THEN
           #qReady := #read.stw.control_ready
           (* *)AND #read.stw.drive_ready
           (* *)AND #read.stw.bus_control;
           #qError := #read.stw.trip
           (* *)OR #read.stw.error_no_trip;
           #qIn_auto := #read.stw.bus_control;
           #qIn_operation := #read.stw.in_operation;
           #qOutput_percent := INT_TO_REAL(#read.man) / 16#4000 * 100;
       END_IF;

       // Send ctw and ref
       #write.ctw.reset := #iReset;
       #write.ctw.dc_break_NOT := NOT #iDC_break;
       #write.ctw.coast_NOT := NOT #iCost;
       #write.ctw.quick_stop_NOT := NOT #iStop_quick;
       #write.ctw.start := #iRef <> 0;
       #write.ref := REAL_TO_INT(#iRef / 100 * 16#4000);
       #mb_query(mode := #mb_query.c.write.holding_reg,
                 data_addr := 2809,
                 data_ptr := #write);
   END_REGION

   "mb_station_block_footer"(sb := #sb, mb_query := #mb_query);
END_FUNCTION_BLOCK

FUNCTION "p" : UDInt   // FC14, SCL
{ S7_Optimized_Access := 'TRUE' }
VERSION : 0.1
   VAR_INPUT
      "a" : USInt;
      "b" : USInt;
   END_VAR
BEGIN
   // 

   #p := USINT_TO_UDINT(#"a") * 1000
   (* *)+ USINT_TO_UDINT(#"b") * 10
   (* *)- 1;
END_FUNCTION

// folder: Library/Modbus/Station blocks/sb tested/Ponsel mesure

FUNCTION_BLOCK "Ponsel_mesure_Conductivity_C4E"   // FB105, SCL
{ S7_Optimized_Access := 'TRUE' }
VERSION : 0.1
   VAR_INPUT
      mb_addr : UInt := 255;   // 255=broadcast
   END_VAR
   VAR_OUTPUT
      Temperature : Real;   // [degree C]
      Conductivity : Real;   // [uS/cm]
      Salinity : Real;   // [ppt]
      TDS_Kcl : Real;   // [ppm]
      measurement_ok : Bool;
   END_VAR
   VAR_IN_OUT
      mb_query : "mb_query";
   END_VAR
   VAR
      ponsel_mesure : "Ponsel_mesure";
   END_VAR
   VAR_TEMP
      start : Bool;
   END_VAR
BEGIN
   // Ponsel mesure - Conductivity_C4E

   #start := true; // Continuous measurements

   #ponsel_mesure.minimum_measurement_interval := T#1s;
   #ponsel_mesure(mb_addr := #mb_addr,
                  compensate_enable := false,
                  Measurement_ok => #measurement_ok,
                  start_measurement := #start,
                  mb_query := #mb_query);

   #Temperature := #ponsel_mesure.data1.value[0];  // [degree C]
   #Conductivity := #ponsel_mesure.data1.value[1]; // [uS/cm]
   #Salinity := #ponsel_mesure.data1.value[2];     // [ppt]
   #TDS_Kcl := #ponsel_mesure.data1.value[3];      // [ppm]
END_FUNCTION_BLOCK

FUNCTION_BLOCK "Ponsel_mesure_Dissolved_oxygen"   // FB106, SCL
{ S7_Optimized_Access := 'TRUE' }
VERSION : 0.1
   VAR_INPUT
      mb_addr : UInt := 10;   // 255=broadcast
      start : Bool := TRUE;   // (Else use start to init messurements)
      measurement_interval : Time := T#1M;
      compensate_atmospheric_pressure : Real := 1013.0;   // hPa
      compensate_salinity : Real := 0.0;   // ppm
   END_VAR
   VAR_OUTPUT
      Temperature : Real;   // [degree C]
      Oxygen_Sat : Real;   // [%]
      Oxygen_mgl : Real;   // [mg/L]
      Oxygen_ppm : Real;   // [ppm]
      measurement_ok : Bool;
      serial_number : String[32];
   END_VAR
   VAR_IN_OUT
      mb_query : "mb_query";
   END_VAR
   VAR
      ponsel_mesure : "Ponsel_mesure";
   END_VAR
   VAR_TEMP
      start_measurement : Bool;
   END_VAR
BEGIN
   // Aqualabo - Ponsel mesure
   // Dissolved oxygen (OPTOD)
   // 
   // Warning: Each pull for sensor measurement, will reduce the available 
   // life span. Please set the measurement interval to appropriate value.

   #start_measurement := #start; // #measurement_interval will define intervals.

   #ponsel_mesure.minimum_measurement_interval := #measurement_interval;
   #ponsel_mesure.compensate[1] := #compensate_atmospheric_pressure;
   #ponsel_mesure.compensate[2] := #compensate_salinity;
   #ponsel_mesure(mb_addr := #mb_addr,
                  compensate_enable := true,
                  Measurement_ok => #measurement_ok,
                  start_measurement := #start_measurement,
                  mb_query := #mb_query);

   #Temperature := #ponsel_mesure.data1.value[0]; // [degree C]
   #Oxygen_Sat := #ponsel_mesure.data1.value[1];  // [%]
   #Oxygen_mgl := #ponsel_mesure.data1.value[2];  // [mg/l]
   #Oxygen_ppm := #ponsel_mesure.data1.value[3];  // [ppm]

   #serial_number := #ponsel_mesure.data2.serial_number;
END_FUNCTION_BLOCK

// folder: Library/Modbus/Station blocks/sb tested/Ponsel mesure/Misc

FUNCTION_BLOCK "ponselMessure_ChangeMbAddr"   // FB94, SCL
{ S7_Optimized_Access := 'TRUE' }
VERSION : 0.1
   VAR_INPUT
      current_addr : USInt;
      new_addr : UInt;
      exec : Bool := TRUE;
   END_VAR
   VAR_OUTPUT
      Done : Bool;
      Error : Bool;
   END_VAR
   VAR_IN_OUT
      mb_query : "mb_query";
   END_VAR
   VAR_TEMP
      d : Bool;
      "e" : Bool;
   END_VAR
BEGIN
   IF #new_addr < 1 OR #new_addr > 247
       OR #new_addr = #current_addr
   THEN
       #"e" := TRUE;
   ELSIF #exec THEN
       #mb_query(mb_addr := #current_addr,
                 mode := #mb_query.c.write.holding_reg,
                 data_addr := 16#A3,
                 Done => #d,
                 Error => #"e",
                 data_ptr := #new_addr);
   END_IF;
   #Done := #d;
   #Error := #"e";
END_FUNCTION_BLOCK

